LIN {X 0,Y 212.666,Z 436.056,A -85,B 0,C 180,E1 -21906.919,E2 -21906.919} C_VEL
LIN {X 0,Y 215.968,Z 426.694,A -85,B 0,C 180,E1 -21909.087,E2 -21909.087} C_VEL
LIN {X 0,Y 219.252,Z 415.76,A -85,B 0,C 180,E1 -21911.08,E2 -21911.08} C_VEL
LIN {X 0,Y 221.834,Z 405.227,A -85,B 0,C 180,E1 -21912.574,E2 -21912.574} C_VEL
LIN {X 0,Y 224.1,Z 393.658,A -85,B 0,C 180,E1 -21913.837,E2 -21913.837} C_VEL
LIN {X 0,Y 225.668,Z 381.684,A -85,B 0,C 180,E1 -21914.841,E2 -21914.841} C_VEL
LIN {X 0,Y 226.691,Z 369.485,A -85,B 0,C 180,E1 -21915.541,E2 -21915.541} C_VEL
LIN {X 0,Y 228.107,Z 336.25,A -85,B 0,C 180,E1 -21916.66,E2 -21916.66} C_VEL
LIN {X 0,Y 221.645,Z 324.171,A -85,B 0,C 180,E1 -21918.78,E2 -21918.78} C_VEL
LIN {X 0,Y 214.301,Z 312.104,A -85,B 0,C 180,E1 -21921.381,E2 -21921.381} C_VEL
LIN {X 0,Y 208.554,Z 303.596,A -85,B 0,C 180,E1 -21923.598,E2 -21923.598} C_VEL
LIN {X 0,Y 205.749,Z 299.629,A -85,B 0,C 180,E1 -21924.755,E2 -21924.755} C_VEL
LIN {X 0,Y 203.216,Z 296.188,A -85,B 0,C 180,E1 -21925.848,E2 -21925.848} C_VEL
LIN {X 0,Y 200.594,Z 292.5,A -85,B 0,C 180,E1 -21927.048,E2 -21927.048} C_VEL
LIN {X 0,Y 197.526,Z 288.904,A -85,B 0,C 180,E1 -21928.494,E2 -21928.494} C_VEL
LIN {X 0,Y 196.478,Z 286.965,A -85,B 0,C 180,E1 -21929.056,E2 -21929.056} C_VEL
LIN {X 0,Y 193.88,Z 284.765,A -85,B 0,C 180,E1 -21930.338,E2 -21930.338} C_VEL
LIN {X 0,Y 192.729,Z 282.176,A -85,B 0,C 180,E1 -21931.187,E2 -21931.187} C_VEL
LIN {X 0,Y 192.614,Z 281.525,A -85,B 0,C 180,E1 -21931.979,E2 -21931.979} C_VEL
LIN {X 0,Y 192.678,Z 281.429,A -85,B 0,C 180,E1 -21936.344,E2 -21936.344} C_VEL
LIN {X 0,Y 192.731,Z 281.449,A -85,B 0,C 180,E1 -21941.459,E2 -21941.459} C_VEL
LIN {X 0,Y 192.761,Z 281.455,A -85,B 0,C 180,E1 -21945.213,E2 -21945.213} C_VEL
LIN {X 0,Y 192.945,Z 281.435,A -85,B 0,C 180,E1 -21949.566,E2 -21949.566} C_VEL
LIN {X 0,Y 192.961,Z 281.448,A -85,B 0,C 180,E1 -21953.727,E2 -21953.727} C_VEL
LIN {X 0,Y 193.226,Z 281.405,A -85,B 0,C 180,E1 -21957.915,E2 -21957.915} C_VEL
LIN {X 0,Y 193.411,Z 281.384,A -85,B 0,C 180,E1 -21960,E2 -21960} C_VEL
LIN {X 0,Y 192.936,Z 281.449,A -85,B 0,C 180,E1 -21964.177,E2 -21964.177} C_VEL
LIN {X 0,Y 193.019,Z 281.422,A -85,B 0,C 180,E1 -21968.374,E2 -21968.374} C_VEL
LIN {X 0,Y 192.791,Z 281.45,A -85,B 0,C 180,E1 -21972.634,E2 -21972.634} C_VEL
LIN {X 0,Y 192.745,Z 281.468,A -85,B 0,C 180,E1 -21976.959,E2 -21976.959} C_VEL
LIN {X 0,Y 192.607,Z 281.485,A -85,B 0,C 180,E1 -21981.4,E2 -21981.4} C_VEL
LIN {X 0,Y 192.637,Z 281.491,A -85,B 0,C 180,E1 -21984.207,E2 -21984.207} C_VEL
LIN {X 0,Y 192.59,Z 281.62,A -85,B 0,C 180,E1 -21989.237,E2 -21989.237} C_VEL
LIN {X 0,Y 195.024,Z 288.184,A -85,B 0,C 180,E1 -21994.021,E2 -21994.021} C_VEL
LIN {X 0,Y 197.384,Z 295.043,A -85,B 0,C 180,E1 -21998.172,E2 -21998.172} C_VEL
LIN {X 0,Y 200.88,Z 300.852,A -85,B 0,C 180,E1 -21999.925,E2 -21999.925} C_VEL
LIN {X 0,Y 205.909,Z 309.501,A -85,B 0,C 180,E1 -22002.219,E2 -22002.219} C_VEL
LIN {X 0,Y 211.718,Z 320.154,A -85,B 0,C 180,E1 -22004.642,E2 -22004.642} C_VEL
LIN {X 0,Y 218.15,Z 333.803,A -85,B 0,C 180,E1 -22007.132,E2 -22007.132} C_VEL
LIN {X 0,Y 221.255,Z 341.29,A -85,B 0,C 180,E1 -22008.283,E2 -22008.283} C_VEL
LIN {X 0,Y 223.88,Z 365.922,A -85,B 0,C 180,E1 -22010.005,E2 -22010.005} C_VEL
LIN {X 0,Y 225.176,Z 381.652,A -85,B 0,C 180,E1 -22010.974,E2 -22010.974} C_VEL
LIN {X 0,Y 225.14,Z 385.521,A -85,B 0,C 180,E1 -22011.123,E2 -22011.123} C_VEL
LIN {X 0,Y 224.591,Z 389.408,A -85,B 0,C 180,E1 -22011.15,E2 -22011.15} C_VEL
LIN {X 0,Y 222.563,Z 397.072,A -85,B 0,C 180,E1 -22010.993,E2 -22010.993} C_VEL
LIN {X 0,Y 219.634,Z 406.689,A -85,B 0,C 180,E1 -22010.771,E2 -22010.771} C_VEL
LIN {X 0,Y 218.506,Z 412.571,A -85,B 0,C 180,E1 -22010.868,E2 -22010.868} C_VEL
LIN {X 0,Y 216.715,Z 425.149,A -85,B 0,C 180,E1 -22011.544,E2 -22011.544} C_VEL
LIN {X 0,Y 214.369,Z 437.19,A -85,B 0,C 180,E1 -22012.514,E2 -22012.514} C_VEL
LIN {X 0,Y 211.274,Z 449.041,A -85,B 0,C 180,E1 -22013.811,E2 -22013.811} C_VEL
LIN {X 0,Y 207.43,Z 460.468,A -85,B 0,C 180,E1 -22015.423,E2 -22015.423} C_VEL
LIN {X 0,Y 203.471,Z 470.808,A -85,B 0,C 180,E1 -22017.337,E2 -22017.337} C_VEL
LIN {X 0,Y 199.84,Z 479.297,A -85,B 0,C 180,E1 -22019.34,E2 -22019.34} C_VEL
LIN {X 0,Y 195.583,Z 488.554,A -85,B 0,C 180,E1 -22022.151,E2 -22022.151} C_VEL
LIN {X 0,Y 191.938,Z 496.066,A -85,B 0,C 180,E1 -22025.097,E2 -22025.097} C_VEL
LIN {X 0,Y 189.021,Z 502.163,A -85,B 0,C 180,E1 -22028.172,E2 -22028.172} C_VEL
LIN {X 0,Y 186.746,Z 507.041,A -85,B 0,C 180,E1 -22031.343,E2 -22031.343} C_VEL
LIN {X 0,Y 185.142,Z 510.839,A -85,B 0,C 180,E1 -22034.59,E2 -22034.59} C_VEL
LIN {X 0,Y 184.418,Z 512.843,A -85,B 0,C 180,E1 -22036.781,E2 -22036.781} C_VEL
LIN {X 0,Y 183.924,Z 515.566,A -85,B 0,C 180,E1 -22041.207,E2 -22041.207} C_VEL
LIN {X 0,Y 184.069,Z 516.35,A -85,B 0,C 180,E1 -22043.422,E2 -22043.422} C_VEL
LIN {X 0,Y 184.377,Z 516.743,A -85,B 0,C 180,E1 -22045.627,E2 -22045.627} C_VEL
LIN {X 0,Y 184.782,Z 516.697,A -85,B 0,C 180,E1 -22047.819,E2 -22047.819} C_VEL
LIN {X 0,Y 184.966,Z 516.195,A -85,B 0,C 180,E1 -22049.999,E2 -22049.999} C_VEL
LIN {X 0,Y 184.839,Z 515.234,A -85,B 0,C 180,E1 -22052.178,E2 -22052.178} C_VEL
LIN {X 0,Y 184.476,Z 513.812,A -85,B 0,C 180,E1 -22054.369,E2 -22054.369} C_VEL
LIN {X 0,Y 184.149,Z 511.34,A -85,B 0,C 180,E1 -22057.124,E2 -22057.124} C_VEL
LIN {X 0,Y 184.126,Z 506.671,A -85,B 0,C 180,E1 -22061.001,E2 -22061.001} C_VEL
LIN {X 0,Y 184.943,Z 500.384,A -85,B 0,C 180,E1 -22064.862,E2 -22064.862} C_VEL
LIN {X 0,Y 186.225,Z 493.516,A -85,B 0,C 180,E1 -22068.139,E2 -22068.139} C_VEL
LIN {X 0,Y 188.344,Z 485.062,A -85,B 0,C 180,E1 -22071.332,E2 -22071.332} C_VEL
LIN {X 0,Y 190.565,Z 476.381,A -85,B 0,C 180,E1 -22073.932,E2 -22073.932} C_VEL
LIN {X 0,Y 192.892,Z 466.861,A -85,B 0,C 180,E1 -22076.215,E2 -22076.215} C_VEL
LIN {X 0,Y 195.38,Z 456.548,A -85,B 0,C 180,E1 -22078.17,E2 -22078.17} C_VEL
LIN {X 0,Y 197.726,Z 445.275,A -85,B 0,C 180,E1 -22079.841,E2 -22079.841} C_VEL
LIN {X 0,Y 199.823,Z 432.646,A -85,B 0,C 180,E1 -22081.248,E2 -22081.248} C_VEL
LIN {X 0,Y 201.398,Z 419.7,A -85,B 0,C 180,E1 -22082.25,E2 -22082.25} C_VEL
LIN {X 0,Y 202.32,Z 405.805,A -85,B 0,C 180,E1 -22082.937,E2 -22082.937} C_VEL
LIN {X 0,Y 203.183,Z 381.621,A -85,B 0,C 180,E1 -22083.764,E2 -22083.764} C_VEL
LIN {X 0,Y 200.75,Z 344.71,A -85,B 0,C 180,E1 -22085.66,E2 -22085.66} C_VEL
LIN {X 0,Y 198.453,Z 320.123,A -85,B 0,C 180,E1 -22087.091,E2 -22087.091} C_VEL
LIN {X 0,Y 192.76,Z 305.892,A -85,B 0,C 180,E1 -22088.801,E2 -22088.801} C_VEL
LIN {X 0,Y 190.025,Z 299.446,A -85,B 0,C 180,E1 -22089.732,E2 -22089.732} C_VEL
LIN {X 0,Y 187.903,Z 291.059,A -85,B 0,C 180,E1 -22093.323,E2 -22093.323} C_VEL
LIN {X 0,Y 185.455,Z 282.487,A -85,B 0,C 180,E1 -22097.48,E2 -22097.48} C_VEL
LIN {X 0,Y 185.495,Z 282.366,A -85,B 0,C 180,E1 -22102.713,E2 -22102.713} C_VEL
LIN {X 0,Y 185.524,Z 282.35,A -85,B 0,C 180,E1 -22107.972,E2 -22107.972} C_VEL
LIN {X 0,Y 185.541,Z 282.371,A -85,B 0,C 180,E1 -22110.595,E2 -22110.595} C_VEL
LIN {X 0,Y 185.574,Z 282.351,A -85,B 0,C 180,E1 -22115.381,E2 -22115.381} C_VEL
LIN {X 0,Y 185.618,Z 282.342,A -85,B 0,C 180,E1 -22121.179,E2 -22121.179} C_VEL
LIN {X 0,Y 185.656,Z 282.353,A -85,B 0,C 180,E1 -22124.634,E2 -22124.634} C_VEL
LIN {X 0,Y 185.881,Z 282.307,A -85,B 0,C 180,E1 -22129.419,E2 -22129.419} C_VEL
LIN {X 0,Y 185.921,Z 282.323,A -85,B 0,C 180,E1 -22133.489,E2 -22133.489} C_VEL
LIN {X 0,Y 186.168,Z 282.272,A -85,B 0,C 180,E1 -22137.837,E2 -22137.837} C_VEL
LIN {X 0,Y 186.37,Z 282.242,A -85,B 0,C 180,E1 -22140,E2 -22140} C_VEL
LIN {X 0,Y 185.867,Z 282.333,A -85,B 0,C 180,E1 -22144.338,E2 -22144.338} C_VEL
LIN {X 0,Y 185.961,Z 282.291,A -85,B 0,C 180,E1 -22148.695,E2 -22148.695} C_VEL
LIN {X 0,Y 185.707,Z 282.35,A -85,B 0,C 180,E1 -22153.125,E2 -22153.125} C_VEL
LIN {X 0,Y 185.646,Z 282.33,A -85,B 0,C 180,E1 -22157.63,E2 -22157.63} C_VEL
LIN {X 0,Y 185.541,Z 282.373,A -85,B 0,C 180,E1 -22162.259,E2 -22162.259} C_VEL
LIN {X 0,Y 185.484,Z 282.36,A -85,B 0,C 180,E1 -22167.045,E2 -22167.045} C_VEL
LIN {X 0,Y 185.525,Z 282.363,A -85,B 0,C 180,E1 -22172.029,E2 -22172.029} C_VEL
LIN {X 0,Y 185.496,Z 282.38,A -85,B 0,C 180,E1 -22177.316,E2 -22177.316} C_VEL
LIN {X 0,Y 185.457,Z 282.336,A -85,B 0,C 180,E1 -22180.722,E2 -22180.722} C_VEL
LIN {X 0,Y 185.452,Z 282.349,A -85,B 0,C 180,E1 -22186.058,E2 -22186.058} C_VEL
LIN {X 0,Y 185.454,Z 282.367,A -85,B 0,C 180,E1 -22189.894,E2 -22189.894} C_VEL
LIN {X 0,Y 185.499,Z 282.332,A -85,B 0,C 180,E1 -22192.716,E2 -22192.716} C_VEL
LIN {X 0,Y 185.528,Z 282.48,A -85,B 0,C 180,E1 -22197.974,E2 -22197.974} C_VEL
LIN {X 0,Y 185.696,Z 283.33,A -85,B 0,C 180,E1 -22198.372,E2 -22198.372} C_VEL
LIN {X 0,Y 187.12,Z 286.075,A -85,B 0,C 180,E1 -22198.87,E2 -22198.87} C_VEL
LIN {X 0,Y 190.505,Z 291.53,A -85,B 0,C 180,E1 -22199.867,E2 -22199.867} C_VEL
LIN {X 0,Y 196.709,Z 302.532,A -85,B 0,C 180,E1 -22201.62,E2 -22201.62} C_VEL
LIN {X 0,Y 203.781,Z 317.099,A -85,B 0,C 180,E1 -22203.532,E2 -22203.532} C_VEL
LIN {X 0,Y 205.564,Z 321.268,A -85,B 0,C 180,E1 -22204.008,E2 -22204.008} C_VEL
LIN {X 0,Y 204.008,Z 369.15,A -85,B 0,C 180,E1 -22205.719,E2 -22205.719} C_VEL
LIN {X 0,Y 203.326,Z 380.674,A -85,B 0,C 180,E1 -22206.445,E2 -22206.445} C_VEL
LIN {X 0,Y 202.053,Z 393.603,A -85,B 0,C 180,E1 -22207.641,E2 -22207.641} C_VEL
LIN {X 0,Y 200.279,Z 405.935,A -85,B 0,C 180,E1 -22209.19,E2 -22209.19} C_VEL
LIN {X 0,Y 198.141,Z 417.489,A -85,B 0,C 180,E1 -22211.117,E2 -22211.117} C_VEL
LIN {X 0,Y 195.987,Z 427.846,A -85,B 0,C 180,E1 -22213.33,E2 -22213.33} C_VEL
LIN {X 0,Y 193.789,Z 437.202,A -85,B 0,C 180,E1 -22215.831,E2 -22215.831} C_VEL
LIN {X 0,Y 191.383,Z 446.228,A -85,B 0,C 180,E1 -22218.885,E2 -22218.885} C_VEL
LIN {X 0,Y 189.347,Z 453.509,A -85,B 0,C 180,E1 -22222,E2 -22222} C_VEL
LIN {X 0,Y 187.582,Z 460.199,A -85,B 0,C 180,E1 -22225.704,E2 -22225.704} C_VEL
LIN {X 0,Y 186.487,Z 464.627,A -85,B 0,C 180,E1 -22228.921,E2 -22228.921} C_VEL
LIN {X 0,Y 185.647,Z 468.025,A -85,B 0,C 180,E1 -22232.17,E2 -22232.17} C_VEL
LIN {X 0,Y 185.454,Z 470.993,A -85,B 0,C 180,E1 -22236.529,E2 -22236.529} C_VEL
LIN {X 0,Y 185.694,Z 472.291,A -85,B 0,C 180,E1 -22240.25,E2 -22240.25} C_VEL
LIN {X 0,Y 186.169,Z 472.505,A -85,B 0,C 180,E1 -22243.092,E2 -22243.092} C_VEL
LIN {X 0,Y 187.574,Z 471.565,A -85,B 0,C 180,E1 -22247.443,E2 -22247.443} C_VEL
LIN {X 0,Y 188.562,Z 470.463,A -85,B 0,C 180,E1 -22249.6,E2 -22249.6} C_VEL
LIN {X 0,Y 190.407,Z 468.162,A -85,B 0,C 180,E1 -22252.665,E2 -22252.665} C_VEL
LIN {X 0,Y 192.795,Z 464.602,A -85,B 0,C 180,E1 -22255.941,E2 -22255.941} C_VEL
LIN {X 0,Y 195.549,Z 460.037,A -85,B 0,C 180,E1 -22259.025,E2 -22259.025} C_VEL
LIN {X 0,Y 199.375,Z 453.086,A -85,B 0,C 180,E1 -22262.518,E2 -22262.518} C_VEL
LIN {X 0,Y 203.086,Z 445.472,A -85,B 0,C 180,E1 -22265.426,E2 -22265.426} C_VEL
LIN {X 0,Y 206.92,Z 436.495,A -85,B 0,C 180,E1 -22268.074,E2 -22268.074} C_VEL
LIN {X 0,Y 210.426,Z 426.876,A -85,B 0,C 180,E1 -22270.324,E2 -22270.324} C_VEL
LIN {X 0,Y 213.492,Z 417.125,A -85,B 0,C 180,E1 -22272.123,E2 -22272.123} C_VEL
LIN {X 0,Y 216.14,Z 406.913,A -85,B 0,C 180,E1 -22273.623,E2 -22273.623} C_VEL
LIN {X 0,Y 218.749,Z 394.311,A -85,B 0,C 180,E1 -22275.022,E2 -22275.022} C_VEL
LIN {X 0,Y 220.418,Z 381.923,A -85,B 0,C 180,E1 -22276.072,E2 -22276.072} C_VEL
LIN {X 0,Y 221.447,Z 369.834,A -85,B 0,C 180,E1 -22276.763,E2 -22276.763} C_VEL
LIN {X 0,Y 222.794,Z 338.838,A -85,B 0,C 180,E1 -22277.833,E2 -22277.833} C_VEL
LIN {X 0,Y 216.755,Z 327.518,A -85,B 0,C 180,E1 -22279.939,E2 -22279.939} C_VEL
LIN {X 0,Y 210.199,Z 316.66,A -85,B 0,C 180,E1 -22282.396,E2 -22282.396} C_VEL
LIN {X 0,Y 204.778,Z 308.452,A -85,B 0,C 180,E1 -22284.608,E2 -22284.608} C_VEL
LIN {X 0,Y 200.168,Z 301.967,A -85,B 0,C 180,E1 -22286.653,E2 -22286.653} C_VEL
LIN {X 0,Y 196.875,Z 297.515,A -85,B 0,C 180,E1 -22288.227,E2 -22288.227} C_VEL
LIN {X 0,Y 194.242,Z 294.054,A -85,B 0,C 180,E1 -22289.565,E2 -22289.565} C_VEL
LIN {X 0,Y 193.394,Z 292.857,A -85,B 0,C 180,E1 -22290.02,E2 -22290.02} C_VEL
LIN {X 0,Y 191.007,Z 290.431,A -85,B 0,C 180,E1 -22291.287,E2 -22291.287} C_VEL
LIN {X 0,Y 189.674,Z 287.958,A -85,B 0,C 180,E1 -22292.108,E2 -22292.108} C_VEL
LIN {X 0,Y 187.145,Z 286.062,A -85,B 0,C 180,E1 -22293.545,E2 -22293.545} C_VEL
LIN {X 0,Y 185.716,Z 283.299,A -85,B 0,C 180,E1 -22294.62,E2 -22294.62} C_VEL
LIN {X 0,Y 185.594,Z 282.426,A -85,B 0,C 180,E1 -22295.486,E2 -22295.486} C_VEL
LIN {X 0,Y 185.673,Z 282.318,A -85,B 0,C 180,E1 -22301.135,E2 -22301.135} C_VEL
LIN {X 0,Y 185.693,Z 282.337,A -85,B 0,C 180,E1 -22304.636,E2 -22304.636} C_VEL
LIN {X 0,Y 185.888,Z 282.315,A -85,B 0,C 180,E1 -22309.419,E2 -22309.419} C_VEL
LIN {X 0,Y 185.926,Z 282.326,A -85,B 0,C 180,E1 -22313.488,E2 -22313.488} C_VEL
LIN {X 0,Y 186.172,Z 282.282,A -85,B 0,C 180,E1 -22317.836,E2 -22317.836} C_VEL
LIN {X 0,Y 186.377,Z 282.26,A -85,B 0,C 180,E1 -22320,E2 -22320} C_VEL
LIN {X 0,Y 185.884,Z 282.329,A -85,B 0,C 180,E1 -22324.336,E2 -22324.336} C_VEL
LIN {X 0,Y 185.969,Z 282.302,A -85,B 0,C 180,E1 -22328.694,E2 -22328.694} C_VEL
LIN {X 0,Y 185.718,Z 282.33,A -85,B 0,C 180,E1 -22333.123,E2 -22333.123} C_VEL
LIN {X 0,Y 185.682,Z 282.344,A -85,B 0,C 180,E1 -22337.625,E2 -22337.625} C_VEL
LIN {X 0,Y 185.569,Z 282.36,A -85,B 0,C 180,E1 -22342.254,E2 -22342.254} C_VEL
LIN {X 0,Y 185.545,Z 282.567,A -85,B 0,C 180,E1 -22346.426,E2 -22346.426} C_VEL
LIN {X 0,Y 187.951,Z 288.856,A -85,B 0,C 180,E1 -22351.567,E2 -22351.567} C_VEL
LIN {X 0,Y 189.577,Z 293.321,A -85,B 0,C 180,E1 -22354.556,E2 -22354.556} C_VEL
LIN {X 0,Y 193.718,Z 299.814,A -85,B 0,C 180,E1 -22356.944,E2 -22356.944} C_VEL
LIN {X 0,Y 199.001,Z 308.663,A -85,B 0,C 180,E1 -22359.669,E2 -22359.669} C_VEL
LIN {X 0,Y 202.611,Z 315.139,A -85,B 0,C 180,E1 -22361.383,E2 -22361.383} C_VEL
LIN {X 0,Y 207.767,Z 324.854,A -85,B 0,C 180,E1 -22363.652,E2 -22363.652} C_VEL
LIN {X 0,Y 213.978,Z 338.398,A -85,B 0,C 180,E1 -22366.198,E2 -22366.198} C_VEL
LIN {X 0,Y 216.453,Z 344.843,A -85,B 0,C 180,E1 -22367.187,E2 -22367.187} C_VEL
LIN {X 0,Y 218.786,Z 368.364,A -85,B 0,C 180,E1 -22368.869,E2 -22368.869} C_VEL
LIN {X 0,Y 220.155,Z 387.448,A -85,B 0,C 180,E1 -22370.049,E2 -22370.049} C_VEL
LIN {X 0,Y 218.626,Z 411.388,A -85,B 0,C 180,E1 -22370.816,E2 -22370.816} C_VEL
LIN {X 0,Y 218.506,Z 412.571,A -85,B 0,C 180,E1 -22370.868,E2 -22370.868} C_VEL
LIN {X 0,Y 217.532,Z 416.438,A -85,B 0,C 180,E1 -22370.922,E2 -22370.922} C_VEL
LIN {X 0,Y 214.526,Z 422.459,A -85,B 0,C 180,E1 -22370.763,E2 -22370.763} C_VEL
LIN {X 0,Y 211.291,Z 428.377,A -85,B 0,C 180,E1 -22370.669,E2 -22370.669} C_VEL
LIN {X 0,Y 209.961,Z 432.081,A -85,B 0,C 180,E1 -22370.846,E2 -22370.846} C_VEL
LIN {X 0,Y 207.055,Z 443.97,A -85,B 0,C 180,E1 -22372.033,E2 -22372.033} C_VEL
LIN {X 0,Y 203.107,Z 456.364,A -85,B 0,C 180,E1 -22373.661,E2 -22373.661} C_VEL
LIN {X 0,Y 198.855,Z 467.265,A -85,B 0,C 180,E1 -22375.564,E2 -22375.564} C_VEL
LIN {X 0,Y 194.521,Z 477.091,A -85,B 0,C 180,E1 -22377.797,E2 -22377.797} C_VEL
LIN {X 0,Y 190.756,Z 485.197,A -85,B 0,C 180,E1 -22380.173,E2 -22380.173} C_VEL
LIN {X 0,Y 186.695,Z 493.199,A -85,B 0,C 180,E1 -22383.145,E2 -22383.145} C_VEL
LIN {X 0,Y 183.406,Z 499.661,A -85,B 0,C 180,E1 -22386.274,E2 -22386.274} C_VEL
LIN {X 0,Y 180.655,Z 504.858,A -85,B 0,C 180,E1 -22389.504,E2 -22389.504} C_VEL
LIN {X 0,Y 178.772,Z 508.973,A -85,B 0,C 180,E1 -22392.851,E2 -22392.851} C_VEL
LIN {X 0,Y 177.443,Z 512.076,A -85,B 0,C 180,E1 -22396.252,E2 -22396.252} C_VEL
LIN {X 0,Y 176.844,Z 514.752,A -85,B 0,C 180,E1 -22400.852,E2 -22400.852} C_VEL
LIN {X 0,Y 177,Z 515.522,A -85,B 0,C 180,E1 -22403.158,E2 -22403.158} C_VEL
LIN {X 0,Y 177.275,Z 515.887,A -85,B 0,C 180,E1 -22405.451,E2 -22405.451} C_VEL
LIN {X 0,Y 177.719,Z 515.816,A -85,B 0,C 180,E1 -22407.733,E2 -22407.733} C_VEL
LIN {X 0,Y 177.919,Z 515.297,A -85,B 0,C 180,E1 -22409.999,E2 -22409.999} C_VEL
LIN {X 0,Y 177.744,Z 514.31,A -85,B 0,C 180,E1 -22412.265,E2 -22412.265} C_VEL
LIN {X 0,Y 177.367,Z 512.856,A -85,B 0,C 180,E1 -22414.544,E2 -22414.544} C_VEL
LIN {X 0,Y 177.023,Z 509.787,A -85,B 0,C 180,E1 -22417.985,E2 -22417.985} C_VEL
LIN {X 0,Y 177.103,Z 505.63,A -85,B 0,C 180,E1 -22421.443,E2 -22421.443} C_VEL
LIN {X 0,Y 178.011,Z 499.269,A -85,B 0,C 180,E1 -22425.454,E2 -22425.454} C_VEL
LIN {X 0,Y 179.436,Z 492.349,A -85,B 0,C 180,E1 -22428.851,E2 -22428.851} C_VEL
LIN {X 0,Y 181.695,Z 483.732,A -85,B 0,C 180,E1 -22432.185,E2 -22432.185} C_VEL
LIN {X 0,Y 184.039,Z 475.033,A -85,B 0,C 180,E1 -22434.837,E2 -22434.837} C_VEL
LIN {X 0,Y 186.439,Z 465.402,A -85,B 0,C 180,E1 -22437.196,E2 -22437.196} C_VEL
LIN {X 0,Y 188.767,Z 456.418,A -85,B 0,C 180,E1 -22438.945,E2 -22438.945} C_VEL
LIN {X 0,Y 191.208,Z 445.319,A -85,B 0,C 180,E1 -22440.661,E2 -22440.661} C_VEL
LIN {X 0,Y 193.38,Z 433.007,A -85,B 0,C 180,E1 -22442.106,E2 -22442.106} C_VEL
LIN {X 0,Y 195.043,Z 420.403,A -85,B 0,C 180,E1 -22443.151,E2 -22443.151} C_VEL
LIN {X 0,Y 196.029,Z 407.345,A -85,B 0,C 180,E1 -22443.859,E2 -22443.859} C_VEL
LIN {X 0,Y 197.053,Z 382.986,A -85,B 0,C 180,E1 -22444.714,E2 -22444.714} C_VEL
LIN {X 0,Y 194.738,Z 345.918,A -85,B 0,C 180,E1 -22446.685,E2 -22446.685} C_VEL
LIN {X 0,Y 192.633,Z 322.522,A -85,B 0,C 180,E1 -22448.097,E2 -22448.097} C_VEL
LIN {X 0,Y 186.404,Z 306.851,A -85,B 0,C 180,E1 -22450.098,E2 -22450.098} C_VEL
LIN {X 0,Y 182.658,Z 298.536,A -85,B 0,C 180,E1 -22451.405,E2 -22451.405} C_VEL
LIN {X 0,Y 180.871,Z 291.89,A -85,B 0,C 180,E1 -22454.378,E2 -22454.378} C_VEL
LIN {X 0,Y 178.422,Z 283.367,A -85,B 0,C 180,E1 -22458.748,E2 -22458.748} C_VEL
LIN {X 0,Y 178.413,Z 283.259,A -85,B 0,C 180,E1 -22463.781,E2 -22463.781} C_VEL
LIN {X 0,Y 178.478,Z 283.23,A -85,B 0,C 180,E1 -22466.545,E2 -22466.545} C_VEL
LIN {X 0,Y 178.437,Z 283.258,A -85,B 0,C 180,E1 -22471.795,E2 -22471.795} C_VEL
LIN {X 0,Y 178.509,Z 283.228,A -85,B 0,C 180,E1 -22474.889,E2 -22474.889} C_VEL
LIN {X 0,Y 178.6,Z 283.213,A -85,B 0,C 180,E1 -22481.651,E2 -22481.651} C_VEL
LIN {X 0,Y 178.634,Z 283.234,A -85,B 0,C 180,E1 -22486.346,E2 -22486.346} C_VEL
LIN {X 0,Y 178.896,Z 283.174,A -85,B 0,C 180,E1 -22490.959,E2 -22490.959} C_VEL
LIN {X 0,Y 179.116,Z 283.15,A -85,B 0,C 180,E1 -22497.752,E2 -22497.752} C_VEL
LIN {X 0,Y 179.335,Z 283.117,A -85,B 0,C 180,E1 -22500,E2 -22500} C_VEL
LIN {X 0,Y 178.816,Z 283.21,A -85,B 0,C 180,E1 -22504.509,E2 -22504.509} C_VEL
LIN {X 0,Y 178.894,Z 283.17,A -85,B 0,C 180,E1 -22509.042,E2 -22509.042} C_VEL
LIN {X 0,Y 178.634,Z 283.232,A -85,B 0,C 180,E1 -22513.655,E2 -22513.655} C_VEL
LIN {X 0,Y 178.549,Z 283.222,A -85,B 0,C 180,E1 -22519.154,E2 -22519.154} C_VEL
LIN {X 0,Y 178.458,Z 283.232,A -85,B 0,C 180,E1 -22525.077,E2 -22525.077} C_VEL
LIN {X 0,Y 178.445,Z 283.255,A -85,B 0,C 180,E1 -22530.798,E2 -22530.798} C_VEL
LIN {X 0,Y 178.478,Z 283.233,A -85,B 0,C 180,E1 -22534.219,E2 -22534.219} C_VEL
LIN {X 0,Y 178.382,Z 283.247,A -85,B 0,C 180,E1 -22539.079,E2 -22539.079} C_VEL
LIN {X 0,Y 178.389,Z 283.198,A -85,B 0,C 180,E1 -22542.049,E2 -22542.049} C_VEL
LIN {X 0,Y 178.388,Z 283.21,A -85,B 0,C 180,E1 -22545.167,E2 -22545.167} C_VEL
LIN {X 0,Y 178.395,Z 283.265,A -85,B 0,C 180,E1 -22548.463,E2 -22548.463} C_VEL
LIN {X 0,Y 178.417,Z 283.216,A -85,B 0,C 180,E1 -22553.784,E2 -22553.784} C_VEL
LIN {X 0,Y 178.519,Z 283.518,A -85,B 0,C 180,E1 -22556.417,E2 -22556.417} C_VEL
LIN {X 0,Y 178.889,Z 284.831,A -85,B 0,C 180,E1 -22556.821,E2 -22556.821} C_VEL
LIN {X 0,Y 180.617,Z 287.486,A -85,B 0,C 180,E1 -22557.401,E2 -22557.401} C_VEL
LIN {X 0,Y 188.928,Z 301.506,A -85,B 0,C 180,E1 -22559.984,E2 -22559.984} C_VEL
LIN {X 0,Y 196.997,Z 317.521,A -85,B 0,C 180,E1 -22562.318,E2 -22562.318} C_VEL
LIN {X 0,Y 199.474,Z 323.359,A -85,B 0,C 180,E1 -22563.024,E2 -22563.024} C_VEL
LIN {X 0,Y 197.795,Z 370.595,A -85,B 0,C 180,E1 -22564.763,E2 -22564.763} C_VEL
LIN {X 0,Y 197.092,Z 381.91,A -85,B 0,C 180,E1 -22565.512,E2 -22565.512} C_VEL
LIN {X 0,Y 195.748,Z 394.738,A -85,B 0,C 180,E1 -22566.74,E2 -22566.74} C_VEL
LIN {X 0,Y 194.04,Z 406.146,A -85,B 0,C 180,E1 -22568.209,E2 -22568.209} C_VEL
LIN {X 0,Y 191.798,Z 417.86,A -85,B 0,C 180,E1 -22570.189,E2 -22570.189} C_VEL
LIN {X 0,Y 189.536,Z 428.297,A -85,B 0,C 180,E1 -22572.467,E2 -22572.467} C_VEL
LIN {X 0,Y 186.986,Z 438.57,A -85,B 0,C 180,E1 -22575.304,E2 -22575.304} C_VEL
LIN {X 0,Y 184.474,Z 447.497,A -85,B 0,C 180,E1 -22578.464,E2 -22578.464} C_VEL
LIN {X 0,Y 182.388,Z 454.701,A -85,B 0,C 180,E1 -22581.693,E2 -22581.693} C_VEL
LIN {X 0,Y 181.06,Z 459.572,A -85,B 0,C 180,E1 -22584.432,E2 -22584.432} C_VEL
LIN {X 0,Y 179.761,Z 464.328,A -85,B 0,C 180,E1 -22587.76,E2 -22587.76} C_VEL
LIN {X 0,Y 178.814,Z 468.004,A -85,B 0,C 180,E1 -22591.127,E2 -22591.127} C_VEL
LIN {X 0,Y 178.423,Z 470.667,A -85,B 0,C 180,E1 -22594.519,E2 -22594.519} C_VEL
LIN {X 0,Y 178.41,Z 471.933,A -85,B 0,C 180,E1 -22596.788,E2 -22596.788} C_VEL
LIN {X 0,Y 178.674,Z 473.139,A -85,B 0,C 180,E1 -22600.464,E2 -22600.464} C_VEL
LIN {X 0,Y 179.237,Z 473.348,A -85,B 0,C 180,E1 -22603.608,E2 -22603.608} C_VEL
LIN {X 0,Y 179.911,Z 473.045,A -85,B 0,C 180,E1 -22605.87,E2 -22605.87} C_VEL
LIN {X 0,Y 180.778,Z 472.346,A -85,B 0,C 180,E1 -22608.121,E2 -22608.121} C_VEL
LIN {X 0,Y 181.855,Z 471.206,A -85,B 0,C 180,E1 -22610.354,E2 -22610.354} C_VEL
LIN {X 0,Y 183.682,Z 469.046,A -85,B 0,C 180,E1 -22613.321,E2 -22613.321} C_VEL
LIN {X 0,Y 186.393,Z 465.236,A -85,B 0,C 180,E1 -22616.902,E2 -22616.902} C_VEL
LIN {X 0,Y 189.323,Z 460.61,A -85,B 0,C 180,E1 -22620.076,E2 -22620.076} C_VEL
LIN {X 0,Y 192.75,Z 454.697,A -85,B 0,C 180,E1 -22623.157,E2 -22623.157} C_VEL
LIN {X 0,Y 196.6,Z 447.279,A -85,B 0,C 180,E1 -22626.146,E2 -22626.146} C_VEL
LIN {X 0,Y 200.162,Z 439.645,A -85,B 0,C 180,E1 -22628.552,E2 -22628.552} C_VEL
LIN {X 0,Y 203.852,Z 430.268,A -85,B 0,C 180,E1 -22630.923,E2 -22630.923} C_VEL
LIN {X 0,Y 207.415,Z 419.763,A -85,B 0,C 180,E1 -22632.993,E2 -22632.993} C_VEL
LIN {X 0,Y 210.587,Z 408.315,A -85,B 0,C 180,E1 -22634.76,E2 -22634.76} C_VEL
LIN {X 0,Y 213.217,Z 396.321,A -85,B 0,C 180,E1 -22636.142,E2 -22636.142} C_VEL
LIN {X 0,Y 215.028,Z 384.131,A -85,B 0,C 180,E1 -22637.215,E2 -22637.215} C_VEL
LIN {X 0,Y 216.106,Z 373.156,A -85,B 0,C 180,E1 -22637.893,E2 -22637.893} C_VEL
LIN {X 0,Y 217.045,Z 354.634,A -85,B 0,C 180,E1 -22638.597,E2 -22638.597} C_VEL
LIN {X 0,Y 217.556,Z 341.405,A -85,B 0,C 180,E1 -22639.072,E2 -22639.072} C_VEL
LIN {X 0,Y 210.814,Z 328.836,A -85,B 0,C 180,E1 -22641.593,E2 -22641.593} C_VEL
LIN {X 0,Y 202.87,Z 315.926,A -85,B 0,C 180,E1 -22644.862,E2 -22644.862} C_VEL
LIN {X 0,Y 196.87,Z 307.354,A -85,B 0,C 180,E1 -22647.623,E2 -22647.623} C_VEL
LIN {X 0,Y 193.77,Z 303.143,A -85,B 0,C 180,E1 -22649.181,E2 -22649.181} C_VEL
LIN {X 0,Y 190.593,Z 298.893,A -85,B 0,C 180,E1 -22650.898,E2 -22650.898} C_VEL
LIN {X 0,Y 188.022,Z 295.765,A -85,B 0,C 180,E1 -22652.371,E2 -22652.371} C_VEL
LIN {X 0,Y 186.959,Z 294.17,A -85,B 0,C 180,E1 -22653.034,E2 -22653.034} C_VEL
LIN {X 0,Y 184.405,Z 291.722,A -85,B 0,C 180,E1 -22654.611,E2 -22654.611} C_VEL
LIN {X 0,Y 182.865,Z 288.946,A -85,B 0,C 180,E1 -22655.731,E2 -22655.731} C_VEL
LIN {X 0,Y 180.118,Z 286.805,A -85,B 0,C 180,E1 -22657.639,E2 -22657.639} C_VEL
LIN {X 0,Y 178.77,Z 284.422,A -85,B 0,C 180,E1 -22658.826,E2 -22658.826} C_VEL
LIN {X 0,Y 178.582,Z 283.45,A -85,B 0,C 180,E1 -22659.599,E2 -22659.599} C_VEL
LIN {X 0,Y 178.648,Z 283.202,A -85,B 0,C 180,E1 -22661.656,E2 -22661.656} C_VEL
LIN {X 0,Y 178.656,Z 283.214,A -85,B 0,C 180,E1 -22666.347,E2 -22666.347} C_VEL
LIN {X 0,Y 178.903,Z 283.179,A -85,B 0,C 180,E1 -22670.959,E2 -22670.959} C_VEL
LIN {X 0,Y 179.119,Z 283.159,A -85,B 0,C 180,E1 -22677.751,E2 -22677.751} C_VEL
LIN {X 0,Y 179.342,Z 283.135,A -85,B 0,C 180,E1 -22680,E2 -22680} C_VEL
LIN {X 0,Y 178.833,Z 283.209,A -85,B 0,C 180,E1 -22684.508,E2 -22684.508} C_VEL
LIN {X 0,Y 178.901,Z 283.185,A -85,B 0,C 180,E1 -22689.04,E2 -22689.04} C_VEL
LIN {X 0,Y 178.647,Z 283.211,A -85,B 0,C 180,E1 -22693.653,E2 -22693.653} C_VEL
LIN {X 0,Y 178.608,Z 283.23,A -85,B 0,C 180,E1 -22699.202,E2 -22699.202} C_VEL
LIN {X 0,Y 178.543,Z 283.423,A -85,B 0,C 180,E1 -22703.027,E2 -22703.027} C_VEL
LIN {X 0,Y 180.409,Z 288.564,A -85,B 0,C 180,E1 -22707.87,E2 -22707.87} C_VEL
LIN {X 0,Y 181.524,Z 291.333,A -85,B 0,C 180,E1 -22709.979,E2 -22709.979} C_VEL
LIN {X 0,Y 187.109,Z 299.664,A -85,B 0,C 180,E1 -22713.805,E2 -22713.805} C_VEL
LIN {X 0,Y 191.667,Z 307.029,A -85,B 0,C 180,E1 -22716.511,E2 -22716.511} C_VEL
LIN {X 0,Y 196.182,Z 314.871,A -85,B 0,C 180,E1 -22718.935,E2 -22718.935} C_VEL
LIN {X 0,Y 199.235,Z 320.508,A -85,B 0,C 180,E1 -22720.458,E2 -22720.458} C_VEL
LIN {X 0,Y 204.276,Z 330.42,A -85,B 0,C 180,E1 -22722.803,E2 -22722.803} C_VEL
LIN {X 0,Y 209.643,Z 342.407,A -85,B 0,C 180,E1 -22725.13,E2 -22725.13} C_VEL
LIN {X 0,Y 211.607,Z 347.396,A -85,B 0,C 180,E1 -22725.955,E2 -22725.955} C_VEL
LIN {X 0,Y 213.626,Z 368.549,A -85,B 0,C 180,E1 -22727.531,E2 -22727.531} C_VEL
LIN {X 0,Y 214.957,Z 387.567,A -85,B 0,C 180,E1 -22728.762,E2 -22728.762} C_VEL
LIN {X 0,Y 213.467,Z 410.427,A -85,B 0,C 180,E1 -22729.514,E2 -22729.514} C_VEL
LIN {X 0,Y 211.523,Z 424.033,A -85,B 0,C 180,E1 -22730.235,E2 -22730.235} C_VEL
LIN {X 0,Y 209.961,Z 432.081,A -85,B 0,C 180,E1 -22730.846,E2 -22730.846} C_VEL
LIN {X 0,Y 208.104,Z 437.7,A -85,B 0,C 180,E1 -22731.229,E2 -22731.229} C_VEL
LIN {X 0,Y 203.46,Z 446.41,A -85,B 0,C 180,E1 -22731.68,E2 -22731.68} C_VEL
LIN {X 0,Y 198.515,Z 454.585,A -85,B 0,C 180,E1 -22732.307,E2 -22732.307} C_VEL
LIN {X 0,Y 196.189,Z 459.393,A -85,B 0,C 180,E1 -22732.964,E2 -22732.964} C_VEL
LIN {X 0,Y 192.104,Z 469.094,A -85,B 0,C 180,E1 -22734.816,E2 -22734.816} C_VEL
LIN {X 0,Y 187.723,Z 478.412,A -85,B 0,C 180,E1 -22737.122,E2 -22737.122} C_VEL
LIN {X 0,Y 183.128,Z 487.52,A -85,B 0,C 180,E1 -22740.072,E2 -22740.072} C_VEL
LIN {X 0,Y 179.126,Z 494.911,A -85,B 0,C 180,E1 -22743.179,E2 -22743.179} C_VEL
LIN {X 0,Y 175.87,Z 500.897,A -85,B 0,C 180,E1 -22746.446,E2 -22746.446} C_VEL
LIN {X 0,Y 173.241,Z 505.67,A -85,B 0,C 180,E1 -22749.828,E2 -22749.828} C_VEL
LIN {X 0,Y 171.418,Z 509.384,A -85,B 0,C 180,E1 -22753.321,E2 -22753.321} C_VEL
LIN {X 0,Y 170.5,Z 511.305,A -85,B 0,C 180,E1 -22755.68,E2 -22755.68} C_VEL
LIN {X 0,Y 169.79,Z 513.94,A -85,B 0,C 180,E1 -22760.469,E2 -22760.469} C_VEL
LIN {X 0,Y 169.934,Z 514.729,A -85,B 0,C 180,E1 -22763.012,E2 -22763.012} C_VEL
LIN {X 0,Y 170.653,Z 514.935,A -85,B 0,C 180,E1 -22767.639,E2 -22767.639} C_VEL
LIN {X 0,Y 170.872,Z 514.4,A -85,B 0,C 180,E1 -22769.999,E2 -22769.999} C_VEL
LIN {X 0,Y 170.65,Z 513.386,A -85,B 0,C 180,E1 -22772.359,E2 -22772.359} C_VEL
LIN {X 0,Y 170.259,Z 511.892,A -85,B 0,C 180,E1 -22774.734,E2 -22774.734} C_VEL
LIN {X 0,Y 169.946,Z 508.784,A -85,B 0,C 180,E1 -22778.32,E2 -22778.32} C_VEL
LIN {X 0,Y 170.108,Z 504.582,A -85,B 0,C 180,E1 -22781.92,E2 -22781.92} C_VEL
LIN {X 0,Y 171.118,Z 498.155,A -85,B 0,C 180,E1 -22786.094,E2 -22786.094} C_VEL
LIN {X 0,Y 172.676,Z 491.178,A -85,B 0,C 180,E1 -22789.618,E2 -22789.618} C_VEL
LIN {X 0,Y 174.997,Z 482.709,A -85,B 0,C 180,E1 -22792.988,E2 -22792.988} C_VEL
LIN {X 0,Y 177.791,Z 472.674,A -85,B 0,C 180,E1 -22796.087,E2 -22796.087} C_VEL
LIN {X 0,Y 180.504,Z 462.773,A -85,B 0,C 180,E1 -22798.485,E2 -22798.485} C_VEL
LIN {X 0,Y 183.288,Z 451.932,A -85,B 0,C 180,E1 -22800.533,E2 -22800.533} C_VEL
LIN {X 0,Y 185.894,Z 439.746,A -85,B 0,C 180,E1 -22802.275,E2 -22802.275} C_VEL
LIN {X 0,Y 188.017,Z 427.006,A -85,B 0,C 180,E1 -22803.618,E2 -22803.618} C_VEL
LIN {X 0,Y 189.436,Z 414.04,A -85,B 0,C 180,E1 -22804.565,E2 -22804.565} C_VEL
LIN {X 0,Y 190.365,Z 398.289,A -85,B 0,C 180,E1 -22805.234,E2 -22805.234} C_VEL
LIN {X 0,Y 190.911,Z 382.796,A -85,B 0,C 180,E1 -22805.804,E2 -22805.804} C_VEL
LIN {X 0,Y 188.68,Z 346.238,A -85,B 0,C 180,E1 -22807.835,E2 -22807.835} C_VEL
LIN {X 0,Y 186.865,Z 324.85,A -85,B 0,C 180,E1 -22809.172,E2 -22809.172} C_VEL
LIN {X 0,Y 181.1,Z 310.273,A -85,B 0,C 180,E1 -22811.14,E2 -22811.14} C_VEL
LIN {X 0,Y 176.651,Z 300.828,A -85,B 0,C 180,E1 -22812.694,E2 -22812.694} C_VEL
LIN {X 0,Y 174.96,Z 296.948,A -85,B 0,C 180,E1 -22813.485,E2 -22813.485} C_VEL
LIN {X 0,Y 172.399,Z 287.851,A -85,B 0,C 180,E1 -22818.087,E2 -22818.087} C_VEL
LIN {X 0,Y 171.364,Z 284.226,A -85,B 0,C 180,E1 -22820.206,E2 -22820.206} C_VEL
LIN {X 0,Y 171.392,Z 284.129,A -85,B 0,C 180,E1 -22825.092,E2 -22825.092} C_VEL
LIN {X 0,Y 171.402,Z 284.132,A -85,B 0,C 180,E1 -22830.526,E2 -22830.526} C_VEL
LIN {X 0,Y 171.43,Z 284.113,A -85,B 0,C 180,E1 -22835.798,E2 -22835.798} C_VEL
LIN {X 0,Y 171.5,Z 284.1,A -85,B 0,C 180,E1 -22840.863,E2 -22840.863} C_VEL
LIN {X 0,Y 171.548,Z 284.116,A -85,B 0,C 180,E1 -22845.771,E2 -22845.771} C_VEL
LIN {X 0,Y 171.835,Z 284.051,A -85,B 0,C 180,E1 -22850.585,E2 -22850.585} C_VEL
LIN {X 0,Y 171.775,Z 284.087,A -85,B 0,C 180,E1 -22855.307,E2 -22855.307} C_VEL
LIN {X 0,Y 172.3,Z 283.992,A -85,B 0,C 180,E1 -22860.001,E2 -22860.001} C_VEL
LIN {X 0,Y 171.766,Z 284.087,A -85,B 0,C 180,E1 -22864.694,E2 -22864.694} C_VEL
LIN {X 0,Y 171.833,Z 284.05,A -85,B 0,C 180,E1 -22869.417,E2 -22869.417} C_VEL
LIN {X 0,Y 171.549,Z 284.11,A -85,B 0,C 180,E1 -22874.23,E2 -22874.23} C_VEL
LIN {X 0,Y 171.474,Z 284.106,A -85,B 0,C 180,E1 -22879.501,E2 -22879.501} C_VEL
LIN {X 0,Y 171.396,Z 284.109,A -85,B 0,C 180,E1 -22885.57,E2 -22885.57} C_VEL
LIN {X 0,Y 171.401,Z 284.133,A -85,B 0,C 180,E1 -22890.567,E2 -22890.567} C_VEL
LIN {X 0,Y 171.388,Z 284.121,A -85,B 0,C 180,E1 -22895.037,E2 -22895.037} C_VEL
LIN {X 0,Y 171.339,Z 284.127,A -85,B 0,C 180,E1 -22898.803,E2 -22898.803} C_VEL
LIN {X 0,Y 171.314,Z 284.078,A -85,B 0,C 180,E1 -22904.22,E2 -22904.22} C_VEL
LIN {X 0,Y 171.327,Z 284.141,A -85,B 0,C 180,E1 -22908.982,E2 -22908.982} C_VEL
LIN {X 0,Y 171.408,Z 284.203,A -85,B 0,C 180,E1 -22914.274,E2 -22914.274} C_VEL
LIN {X 0,Y 171.625,Z 285.187,A -85,B 0,C 180,E1 -22914.861,E2 -22914.861} C_VEL
LIN {X 0,Y 173.121,Z 287.937,A -85,B 0,C 180,E1 -22915.472,E2 -22915.472} C_VEL
LIN {X 0,Y 174.158,Z 289.134,A -85,B 0,C 180,E1 -22915.818,E2 -22915.818} C_VEL
LIN {X 0,Y 183.037,Z 304.018,A -85,B 0,C 180,E1 -22918.786,E2 -22918.786} C_VEL
LIN {X 0,Y 190.781,Z 319.209,A -85,B 0,C 180,E1 -22921.172,E2 -22921.172} C_VEL
LIN {X 0,Y 193.439,Z 325.353,A -85,B 0,C 180,E1 -22921.973,E2 -22921.973} C_VEL
LIN {X 0,Y 191.716,Z 371.101,A -85,B 0,C 180,E1 -22923.697,E2 -22923.697} C_VEL
LIN {X 0,Y 190.981,Z 382.401,A -85,B 0,C 180,E1 -22924.455,E2 -22924.455} C_VEL
LIN {X 0,Y 189.658,Z 394.757,A -85,B 0,C 180,E1 -22925.655,E2 -22925.655} C_VEL
LIN {X 0,Y 187.86,Z 406.345,A -85,B 0,C 180,E1 -22927.163,E2 -22927.163} C_VEL
LIN {X 0,Y 185.797,Z 416.916,A -85,B 0,C 180,E1 -22928.941,E2 -22928.941} C_VEL
LIN {X 0,Y 183.38,Z 427.698,A -85,B 0,C 180,E1 -22931.28,E2 -22931.28} C_VEL
LIN {X 0,Y 180.662,Z 438.245,A -85,B 0,C 180,E1 -22934.2,E2 -22934.2} C_VEL
LIN {X 0,Y 178.447,Z 446.039,A -85,B 0,C 180,E1 -22936.913,E2 -22936.913} C_VEL
LIN {X 0,Y 176.119,Z 453.682,A -85,B 0,C 180,E1 -22940.237,E2 -22940.237} C_VEL
LIN {X 0,Y 174.05,Z 460.7,A -85,B 0,C 180,E1 -22944.207,E2 -22944.207} C_VEL
LIN {X 0,Y 172.702,Z 465.399,A -85,B 0,C 180,E1 -22947.669,E2 -22947.669} C_VEL
LIN {X 0,Y 171.751,Z 469.019,A -85,B 0,C 180,E1 -22951.173,E2 -22951.173} C_VEL
LIN {X 0,Y 171.375,Z 471.629,A -85,B 0,C 180,E1 -22954.705,E2 -22954.705} C_VEL
LIN {X 0,Y 171.371,Z 472.873,A -85,B 0,C 180,E1 -22957.068,E2 -22957.068} C_VEL
LIN {X 0,Y 171.653,Z 473.986,A -85,B 0,C 180,E1 -22960.69,E2 -22960.69} C_VEL
LIN {X 0,Y 172.312,Z 474.193,A -85,B 0,C 180,E1 -22964.166,E2 -22964.166} C_VEL
LIN {X 0,Y 173.051,Z 473.866,A -85,B 0,C 180,E1 -22966.517,E2 -22966.517} C_VEL
LIN {X 0,Y 174.017,Z 473.115,A -85,B 0,C 180,E1 -22968.851,E2 -22968.851} C_VEL
LIN {X 0,Y 176.619,Z 470.375,A -85,B 0,C 180,E1 -22973.449,E2 -22973.449} C_VEL
LIN {X 0,Y 179.081,Z 467.18,A -85,B 0,C 180,E1 -22976.828,E2 -22976.828} C_VEL
LIN {X 0,Y 182.072,Z 462.888,A -85,B 0,C 180,E1 -22980.12,E2 -22980.12} C_VEL
LIN {X 0,Y 185.686,Z 457.179,A -85,B 0,C 180,E1 -22983.41,E2 -22983.41} C_VEL
LIN {X 0,Y 189.458,Z 450.399,A -85,B 0,C 180,E1 -22986.408,E2 -22986.408} C_VEL
LIN {X 0,Y 193.859,Z 441.61,A -85,B 0,C 180,E1 -22989.378,E2 -22989.378} C_VEL
LIN {X 0,Y 197.918,Z 431.997,A -85,B 0,C 180,E1 -22991.931,E2 -22991.931} C_VEL
LIN {X 0,Y 201.37,Z 422.399,A -85,B 0,C 180,E1 -22993.92,E2 -22993.92} C_VEL
LIN {X 0,Y 204.754,Z 411.035,A -85,B 0,C 180,E1 -22995.767,E2 -22995.767} C_VEL
LIN {X 0,Y 207.475,Z 399.747,A -85,B 0,C 180,E1 -22997.171,E2 -22997.171} C_VEL
LIN {X 0,Y 209.662,Z 387.53,A -85,B 0,C 180,E1 -22998.303,E2 -22998.303} C_VEL
LIN {X 0,Y 210.819,Z 376.497,A -85,B 0,C 180,E1 -22999.086,E2 -22999.086} C_VEL
LIN {X 0,Y 211.827,Z 359.602,A -85,B 0,C 180,E1 -22999.788,E2 -22999.788} C_VEL
LIN {X 0,Y 212.534,Z 344.175,A -85,B 0,C 180,E1 -23000.332,E2 -23000.332} C_VEL
LIN {X 0,Y 205.964,Z 331.983,A -85,B 0,C 180,E1 -23002.949,E2 -23002.949} C_VEL
LIN {X 0,Y 199.07,Z 320.682,A -85,B 0,C 180,E1 -23005.974,E2 -23005.974} C_VEL
LIN {X 0,Y 193.976,Z 313.2,A -85,B 0,C 180,E1 -23008.45,E2 -23008.45} C_VEL
LIN {X 0,Y 190.796,Z 308.825,A -85,B 0,C 180,E1 -23010.129,E2 -23010.129} C_VEL
LIN {X 0,Y 187.942,Z 304.917,A -85,B 0,C 180,E1 -23011.752,E2 -23011.752} C_VEL
LIN {X 0,Y 185.191,Z 301.316,A -85,B 0,C 180,E1 -23013.432,E2 -23013.432} C_VEL
LIN {X 0,Y 184.13,Z 300.084,A -85,B 0,C 180,E1 -23014.106,E2 -23014.106} C_VEL
LIN {X 0,Y 181.655,Z 297.193,A -85,B 0,C 180,E1 -23015.769,E2 -23015.769} C_VEL
LIN {X 0,Y 180.475,Z 295.275,A -85,B 0,C 180,E1 -23016.66,E2 -23016.66} C_VEL
LIN {X 0,Y 177.749,Z 292.746,A -85,B 0,C 180,E1 -23018.699,E2 -23018.699} C_VEL
LIN {X 0,Y 176.186,Z 289.976,A -85,B 0,C 180,E1 -23020.106,E2 -23020.106} C_VEL
LIN {X 0,Y 173.09,Z 287.695,A -85,B 0,C 180,E1 -23022.879,E2 -23022.879} C_VEL
LIN {X 0,Y 171.678,Z 284.701,A -85,B 0,C 180,E1 -23024.872,E2 -23024.872} C_VEL
LIN {X 0,Y 171.623,Z 284.122,A -85,B 0,C 180,E1 -23026.38,E2 -23026.38} C_VEL
LIN {X 0,Y 171.842,Z 284.058,A -85,B 0,C 180,E1 -23030.584,E2 -23030.584} C_VEL
LIN {X 0,Y 171.776,Z 284.068,A -85,B 0,C 180,E1 -23035.306,E2 -23035.306} C_VEL
LIN {X 0,Y 172.307,Z 284.01,A -85,B 0,C 180,E1 -23039.999,E2 -23039.999} C_VEL
LIN {X 0,Y 171.783,Z 284.088,A -85,B 0,C 180,E1 -23044.693,E2 -23044.693} C_VEL
LIN {X 0,Y 171.84,Z 284.068,A -85,B 0,C 180,E1 -23049.415,E2 -23049.415} C_VEL
LIN {X 0,Y 171.564,Z 284.096,A -85,B 0,C 180,E1 -23054.228,E2 -23054.228} C_VEL
LIN {X 0,Y 171.609,Z 284.253,A -85,B 0,C 180,E1 -23058.814,E2 -23058.814} C_VEL
LIN {X 0,Y 173.063,Z 288.26,A -85,B 0,C 180,E1 -23063.324,E2 -23063.324} C_VEL
LIN {X 0,Y 179.415,Z 297.758,A -85,B 0,C 180,E1 -23069.237,E2 -23069.237} C_VEL
LIN {X 0,Y 184.486,Z 305.591,A -85,B 0,C 180,E1 -23072.874,E2 -23072.874} C_VEL
LIN {X 0,Y 188.759,Z 312.7,A -85,B 0,C 180,E1 -23075.554,E2 -23075.554} C_VEL
LIN {X 0,Y 192.917,Z 320.152,A -85,B 0,C 180,E1 -23077.918,E2 -23077.918} C_VEL
LIN {X 0,Y 196.339,Z 326.671,A -85,B 0,C 180,E1 -23079.716,E2 -23079.716} C_VEL
LIN {X 0,Y 201.871,Z 338.124,A -85,B 0,C 180,E1 -23082.407,E2 -23082.407} C_VEL
LIN {X 0,Y 206.907,Z 350.295,A -85,B 0,C 180,E1 -23084.695,E2 -23084.695} C_VEL
LIN {X 0,Y 208.697,Z 370.631,A -85,B 0,C 180,E1 -23086.251,E2 -23086.251} C_VEL
LIN {X 0,Y 209.835,Z 389.154,A -85,B 0,C 180,E1 -23087.472,E2 -23087.472} C_VEL
LIN {X 0,Y 208.408,Z 409.715,A -85,B 0,C 180,E1 -23088.162,E2 -23088.162} C_VEL
LIN {X 0,Y 206.331,Z 423.558,A -85,B 0,C 180,E1 -23088.901,E2 -23088.901} C_VEL
LIN {X 0,Y 203.784,Z 435.5,A -85,B 0,C 180,E1 -23089.873,E2 -23089.873} C_VEL
LIN {X 0,Y 200.513,Z 447.34,A -85,B 0,C 180,E1 -23091.206,E2 -23091.206} C_VEL
LIN {X 0,Y 196.189,Z 459.393,A -85,B 0,C 180,E1 -23092.964,E2 -23092.964} C_VEL
LIN {X 0,Y 193.739,Z 464.162,A -85,B 0,C 180,E1 -23093.697,E2 -23093.697} C_VEL
LIN {X 0,Y 188.063,Z 471.482,A -85,B 0,C 180,E1 -23094.771,E2 -23094.771} C_VEL
LIN {X 0,Y 182.235,Z 478.26,A -85,B 0,C 180,E1 -23096.09,E2 -23096.09} C_VEL
LIN {X 0,Y 179.591,Z 482.177,A -85,B 0,C 180,E1 -23097.207,E2 -23097.207} C_VEL
LIN {X 0,Y 174.795,Z 490.858,A -85,B 0,C 180,E1 -23100.492,E2 -23100.492} C_VEL
LIN {X 0,Y 171.522,Z 496.419,A -85,B 0,C 180,E1 -23103.21,E2 -23103.21} C_VEL
LIN {X 0,Y 167.941,Z 502.499,A -85,B 0,C 180,E1 -23107.022,E2 -23107.022} C_VEL
LIN {X 0,Y 165.149,Z 507.516,A -85,B 0,C 180,E1 -23111.387,E2 -23111.387} C_VEL
LIN {X 0,Y 163.578,Z 510.534,A -85,B 0,C 180,E1 -23115.061,E2 -23115.061} C_VEL
LIN {X 0,Y 162.74,Z 513.129,A -85,B 0,C 180,E1 -23120.052,E2 -23120.052} C_VEL
LIN {X 0,Y 162.884,Z 513.927,A -85,B 0,C 180,E1 -23122.925,E2 -23122.925} C_VEL
LIN {X 0,Y 163.584,Z 514.053,A -85,B 0,C 180,E1 -23127.537,E2 -23127.537} C_VEL
LIN {X 0,Y 163.825,Z 513.501,A -85,B 0,C 180,E1 -23129.999,E2 -23129.999} C_VEL
LIN {X 0,Y 163.557,Z 512.461,A -85,B 0,C 180,E1 -23132.462,E2 -23132.462} C_VEL
LIN {X 0,Y 163.151,Z 510.921,A -85,B 0,C 180,E1 -23134.941,E2 -23134.941} C_VEL
LIN {X 0,Y 162.854,Z 507.765,A -85,B 0,C 180,E1 -23138.686,E2 -23138.686} C_VEL
LIN {X 0,Y 163.099,Z 503.517,A -85,B 0,C 180,E1 -23142.441,E2 -23142.441} C_VEL
LIN {X 0,Y 164.219,Z 497.033,A -85,B 0,C 180,E1 -23146.789,E2 -23146.789} C_VEL
LIN {X 0,Y 165.917,Z 490.088,A -85,B 0,C 180,E1 -23150.409,E2 -23150.409} C_VEL
LIN {X 0,Y 168.022,Z 482.87,A -85,B 0,C 180,E1 -23153.411,E2 -23153.411} C_VEL
LIN {X 0,Y 170.582,Z 474.289,A -85,B 0,C 180,E1 -23156.287,E2 -23156.287} C_VEL
LIN {X 0,Y 173.2,Z 464.872,A -85,B 0,C 180,E1 -23158.805,E2 -23158.805} C_VEL
LIN {X 0,Y 175.666,Z 456.12,A -85,B 0,C 180,E1 -23160.668,E2 -23160.668} C_VEL
LIN {X 0,Y 178.3,Z 445.374,A -85,B 0,C 180,E1 -23162.481,E2 -23162.481} C_VEL
LIN {X 0,Y 180.639,Z 433.55,A -85,B 0,C 180,E1 -23164.004,E2 -23164.004} C_VEL
LIN {X 0,Y 182.563,Z 420.878,A -85,B 0,C 180,E1 -23165.185,E2 -23165.185} C_VEL
LIN {X 0,Y 183.713,Z 408.329,A -85,B 0,C 180,E1 -23165.98,E2 -23165.98} C_VEL
LIN {X 0,Y 184.879,Z 383.442,A -85,B 0,C 180,E1 -23166.92,E2 -23166.92} C_VEL
LIN {X 0,Y 182.741,Z 346.763,A -85,B 0,C 180,E1 -23169.042,E2 -23169.042} C_VEL
LIN {X 0,Y 181.169,Z 327.172,A -85,B 0,C 180,E1 -23170.314,E2 -23170.314} C_VEL
LIN {X 0,Y 174.935,Z 311.395,A -85,B 0,C 180,E1 -23172.597,E2 -23172.597} C_VEL
LIN {X 0,Y 169.197,Z 299.746,A -85,B 0,C 180,E1 -23174.763,E2 -23174.763} C_VEL
LIN {X 0,Y 167.415,Z 295.791,A -85,B 0,C 180,E1 -23175.658,E2 -23175.658} C_VEL
LIN {X 0,Y 165,Z 287.343,A -85,B 0,C 180,E1 -23180.29,E2 -23180.29} C_VEL
LIN {X 0,Y 164.339,Z 285.084,A -85,B 0,C 180,E1 -23181.775,E2 -23181.775} C_VEL
LIN {X 0,Y 164.312,Z 284.995,A -85,B 0,C 180,E1 -23186.218,E2 -23186.218} C_VEL
LIN {X 0,Y 164.36,Z 284.99,A -85,B 0,C 180,E1 -23189.129,E2 -23189.129} C_VEL
LIN {X 0,Y 164.387,Z 284.986,A -85,B 0,C 180,E1 -23194.69,E2 -23194.69} C_VEL
LIN {X 0,Y 164.41,Z 284.99,A -85,B 0,C 180,E1 -23200.117,E2 -23200.117} C_VEL
LIN {X 0,Y 164.476,Z 284.994,A -85,B 0,C 180,E1 -23205.145,E2 -23205.145} C_VEL
LIN {X 0,Y 164.756,Z 284.932,A -85,B 0,C 180,E1 -23210.176,E2 -23210.176} C_VEL
LIN {X 0,Y 164.811,Z 284.941,A -85,B 0,C 180,E1 -23212.651,E2 -23212.651} C_VEL
LIN {X 0,Y 165.264,Z 284.867,A -85,B 0,C 180,E1 -23220.001,E2 -23220.001} C_VEL
LIN {X 0,Y 164.807,Z 284.926,A -85,B 0,C 180,E1 -23227.351,E2 -23227.351} C_VEL
LIN {X 0,Y 164.695,Z 284.954,A -85,B 0,C 180,E1 -23231.057,E2 -23231.057} C_VEL
LIN {X 0,Y 164.43,Z 284.97,A -85,B 0,C 180,E1 -23237.41,E2 -23237.41} C_VEL
LIN {X 0,Y 164.414,Z 284.991,A -85,B 0,C 180,E1 -23239.997,E2 -23239.997} C_VEL
LIN {X 0,Y 164.33,Z 284.987,A -85,B 0,C 180,E1 -23246.093,E2 -23246.093} C_VEL
LIN {X 0,Y 164.339,Z 285.007,A -85,B 0,C 180,E1 -23251.211,E2 -23251.211} C_VEL
LIN {X 0,Y 164.276,Z 285.023,A -85,B 0,C 180,E1 -23256.795,E2 -23256.795} C_VEL
LIN {X 0,Y 164.282,Z 284.977,A -85,B 0,C 180,E1 -23259.92,E2 -23259.92} C_VEL
LIN {X 0,Y 164.277,Z 284.947,A -85,B 0,C 180,E1 -23263.344,E2 -23263.344} C_VEL
LIN {X 0,Y 164.257,Z 284.993,A -85,B 0,C 180,E1 -23266.8,E2 -23266.8} C_VEL
LIN {X 0,Y 164.36,Z 285.168,A -85,B 0,C 180,E1 -23272.267,E2 -23272.267} C_VEL
LIN {X 0,Y 164.553,Z 286.07,A -85,B 0,C 180,E1 -23272.781,E2 -23272.781} C_VEL
LIN {X 0,Y 166.037,Z 288.764,A -85,B 0,C 180,E1 -23273.454,E2 -23273.454} C_VEL
LIN {X 0,Y 167.354,Z 290.432,A -85,B 0,C 180,E1 -23273.95,E2 -23273.95} C_VEL
LIN {X 0,Y 169.56,Z 293.727,A -85,B 0,C 180,E1 -23274.781,E2 -23274.781} C_VEL
LIN {X 0,Y 177.917,Z 307.741,A -85,B 0,C 180,E1 -23277.742,E2 -23277.742} C_VEL
LIN {X 0,Y 185.002,Z 321.803,A -85,B 0,C 180,E1 -23280.07,E2 -23280.07} C_VEL
LIN {X 0,Y 187.447,Z 327.188,A -85,B 0,C 180,E1 -23280.843,E2 -23280.843} C_VEL
LIN {X 0,Y 185.716,Z 371.748,A -85,B 0,C 180,E1 -23282.573,E2 -23282.573} C_VEL
LIN {X 0,Y 184.959,Z 382.882,A -85,B 0,C 180,E1 -23283.332,E2 -23283.332} C_VEL
LIN {X 0,Y 183.473,Z 395.89,A -85,B 0,C 180,E1 -23284.627,E2 -23284.627} C_VEL
LIN {X 0,Y 181.421,Z 408.283,A -85,B 0,C 180,E1 -23286.304,E2 -23286.304} C_VEL
LIN {X 0,Y 178.977,Z 419.876,A -85,B 0,C 180,E1 -23288.401,E2 -23288.401} C_VEL
LIN {X 0,Y 176.488,Z 430.257,A -85,B 0,C 180,E1 -23290.822,E2 -23290.822} C_VEL
LIN {X 0,Y 173.914,Z 439.642,A -85,B 0,C 180,E1 -23293.57,E2 -23293.57} C_VEL
LIN {X 0,Y 171.131,Z 448.691,A -85,B 0,C 180,E1 -23296.947,E2 -23296.947} C_VEL
LIN {X 0,Y 168.8,Z 455.984,A -85,B 0,C 180,E1 -23300.415,E2 -23300.415} C_VEL
LIN {X 0,Y 167.045,Z 461.828,A -85,B 0,C 180,E1 -23303.964,E2 -23303.964} C_VEL
LIN {X 0,Y 165.646,Z 466.469,A -85,B 0,C 180,E1 -23307.569,E2 -23307.569} C_VEL
LIN {X 0,Y 164.688,Z 470.034,A -85,B 0,C 180,E1 -23311.224,E2 -23311.224} C_VEL
LIN {X 0,Y 164.33,Z 472.593,A -85,B 0,C 180,E1 -23314.908,E2 -23314.908} C_VEL
LIN {X 0,Y 164.337,Z 473.809,A -85,B 0,C 180,E1 -23317.372,E2 -23317.372} C_VEL
LIN {X 0,Y 164.862,Z 475.004,A -85,B 0,C 180,E1 -23322.308,E2 -23322.308} C_VEL
LIN {X 0,Y 166.228,Z 474.68,A -85,B 0,C 180,E1 -23327.215,E2 -23327.215} C_VEL
LIN {X 0,Y 168.552,Z 472.692,A -85,B 0,C 180,E1 -23332.041,E2 -23332.041} C_VEL
LIN {X 0,Y 170.319,Z 470.806,A -85,B 0,C 180,E1 -23334.795,E2 -23334.795} C_VEL
LIN {X 0,Y 173.724,Z 466.509,A -85,B 0,C 180,E1 -23339.043,E2 -23339.043} C_VEL
LIN {X 0,Y 177.091,Z 461.759,A -85,B 0,C 180,E1 -23342.396,E2 -23342.396} C_VEL
LIN {X 0,Y 180.924,Z 455.715,A -85,B 0,C 180,E1 -23345.639,E2 -23345.639} C_VEL
LIN {X 0,Y 185.241,Z 448.123,A -85,B 0,C 180,E1 -23348.756,E2 -23348.756} C_VEL
LIN {X 0,Y 189.154,Z 440.278,A -85,B 0,C 180,E1 -23351.262,E2 -23351.262} C_VEL
LIN {X 0,Y 193.232,Z 430.643,A -85,B 0,C 180,E1 -23353.713,E2 -23353.713} C_VEL
LIN {X 0,Y 197.153,Z 419.857,A -85,B 0,C 180,E1 -23355.84,E2 -23355.84} C_VEL
LIN {X 0,Y 200.266,Z 409.244,A -85,B 0,C 180,E1 -23357.473,E2 -23357.473} C_VEL
LIN {X 0,Y 202.966,Z 397.832,A -85,B 0,C 180,E1 -23358.805,E2 -23358.805} C_VEL
LIN {X 0,Y 204.867,Z 386.487,A -85,B 0,C 180,E1 -23359.828,E2 -23359.828} C_VEL
LIN {X 0,Y 205.974,Z 376.162,A -85,B 0,C 180,E1 -23360.525,E2 -23360.525} C_VEL
LIN {X 0,Y 207.048,Z 358.485,A -85,B 0,C 180,E1 -23361.242,E2 -23361.242} C_VEL
LIN {X 0,Y 207.521,Z 346.813,A -85,B 0,C 180,E1 -23361.689,E2 -23361.689} C_VEL
LIN {X 0,Y 201.627,Z 335.885,A -85,B 0,C 180,E1 -23364.191,E2 -23364.191} C_VEL
LIN {X 0,Y 195.489,Z 325.646,A -85,B 0,C 180,E1 -23367.059,E2 -23367.059} C_VEL
LIN {X 0,Y 190.627,Z 318.377,A -85,B 0,C 180,E1 -23369.567,E2 -23369.567} C_VEL
LIN {X 0,Y 187.872,Z 314.455,A -85,B 0,C 180,E1 -23371.111,E2 -23371.111} C_VEL
LIN {X 0,Y 185.144,Z 310.716,A -85,B 0,C 180,E1 -23372.748,E2 -23372.748} C_VEL
LIN {X 0,Y 182.111,Z 306.621,A -85,B 0,C 180,E1 -23374.727,E2 -23374.727} C_VEL
LIN {X 0,Y 179.302,Z 303.209,A -85,B 0,C 180,E1 -23376.71,E2 -23376.71} C_VEL
LIN {X 0,Y 178.397,Z 301.7,A -85,B 0,C 180,E1 -23377.43,E2 -23377.43} C_VEL
LIN {X 0,Y 175.783,Z 299.096,A -85,B 0,C 180,E1 -23379.494,E2 -23379.494} C_VEL
LIN {X 0,Y 174.298,Z 296.577,A -85,B 0,C 180,E1 -23380.885,E2 -23380.885} C_VEL
LIN {X 0,Y 171.413,Z 294.217,A -85,B 0,C 180,E1 -23383.627,E2 -23383.627} C_VEL
LIN {X 0,Y 169.797,Z 291.179,A -85,B 0,C 180,E1 -23385.62,E2 -23385.62} C_VEL
LIN {X 0,Y 166.691,Z 289.014,A -85,B 0,C 180,E1 -23389.733,E2 -23389.733} C_VEL
LIN {X 0,Y 165.129,Z 286.35,A -85,B 0,C 180,E1 -23392.894,E2 -23392.894} C_VEL
LIN {X 0,Y 164.824,Z 285.435,A -85,B 0,C 180,E1 -23394.494,E2 -23394.494} C_VEL
LIN {X 0,Y 165.018,Z 284.953,A -85,B 0,C 180,E1 -23397.559,E2 -23397.559} C_VEL
LIN {X 0,Y 165.271,Z 284.886,A -85,B 0,C 180,E1 -23399.999,E2 -23399.999} C_VEL
LIN {X 0,Y 164.817,Z 284.96,A -85,B 0,C 180,E1 -23407.349,E2 -23407.349} C_VEL
LIN {X 0,Y 164.748,Z 285.234,A -85,B 0,C 180,E1 -23411.142,E2 -23411.142} C_VEL
LIN {X 0,Y 164.9,Z 286.468,A -85,B 0,C 180,E1 -23413.086,E2 -23413.086} C_VEL
LIN {X 0,Y 166.404,Z 289.009,A -85,B 0,C 180,E1 -23416.248,E2 -23416.248} C_VEL
LIN {X 0,Y 168.101,Z 290.548,A -85,B 0,C 180,E1 -23418.747,E2 -23418.747} C_VEL
LIN {X 0,Y 171.542,Z 295.328,A -85,B 0,C 180,E1 -23422.985,E2 -23422.985} C_VEL
LIN {X 0,Y 177.287,Z 304.088,A -85,B 0,C 180,E1 -23428.405,E2 -23428.405} C_VEL
LIN {X 0,Y 181.837,Z 311.328,A -85,B 0,C 180,E1 -23431.857,E2 -23431.857} C_VEL
LIN {X 0,Y 185.877,Z 318.339,A -85,B 0,C 180,E1 -23434.551,E2 -23434.551} C_VEL
LIN {X 0,Y 189.924,Z 325.792,A -85,B 0,C 180,E1 -23436.984,E2 -23436.984} C_VEL
LIN {X 0,Y 194.501,Z 334.97,A -85,B 0,C 180,E1 -23439.497,E2 -23439.497} C_VEL
LIN {X 0,Y 199.3,Z 345.757,A -85,B 0,C 180,E1 -23441.933,E2 -23441.933} C_VEL
LIN {X 0,Y 202.405,Z 353.635,A -85,B 0,C 180,E1 -23443.431,E2 -23443.431} C_VEL
LIN {X 0,Y 204.079,Z 375.121,A -85,B 0,C 180,E1 -23445.094,E2 -23445.094} C_VEL
LIN {X 0,Y 204.832,Z 390.378,A -85,B 0,C 180,E1 -23446.098,E2 -23446.098} C_VEL
LIN {X 0,Y 203.361,Z 409.865,A -85,B 0,C 180,E1 -23446.775,E2 -23446.775} C_VEL
LIN {X 0,Y 201.285,Z 423.029,A -85,B 0,C 180,E1 -23447.497,E2 -23447.497} C_VEL
LIN {X 0,Y 198.671,Z 434.669,A -85,B 0,C 180,E1 -23448.449,E2 -23448.449} C_VEL
LIN {X 0,Y 195.032,Z 447.29,A -85,B 0,C 180,E1 -23449.9,E2 -23449.9} C_VEL
LIN {X 0,Y 190.823,Z 458.563,A -85,B 0,C 180,E1 -23451.574,E2 -23451.574} C_VEL
LIN {X 0,Y 186.345,Z 468.749,A -85,B 0,C 180,E1 -23453.558,E2 -23453.558} C_VEL
LIN {X 0,Y 181.784,Z 477.964,A -85,B 0,C 180,E1 -23455.903,E2 -23455.903} C_VEL
LIN {X 0,Y 179.591,Z 482.177,A -85,B 0,C 180,E1 -23457.207,E2 -23457.207} C_VEL
LIN {X 0,Y 176.964,Z 485.954,A -85,B 0,C 180,E1 -23458.424,E2 -23458.424} C_VEL
LIN {X 0,Y 171.131,Z 491.533,A -85,B 0,C 180,E1 -23460.34,E2 -23460.34} C_VEL
LIN {X 0,Y 165.448,Z 496.456,A -85,B 0,C 180,E1 -23462.529,E2 -23462.529} C_VEL
LIN {X 0,Y 163.113,Z 499.152,A -85,B 0,C 180,E1 -23464.146,E2 -23464.146} C_VEL
LIN {X 0,Y 159.864,Z 504.271,A -85,B 0,C 180,E1 -23468.057,E2 -23468.057} C_VEL
LIN {X 0,Y 157.746,Z 507.91,A -85,B 0,C 180,E1 -23471.827,E2 -23471.827} C_VEL
LIN {X 0,Y 156.027,Z 511.233,A -85,B 0,C 180,E1 -23476.984,E2 -23476.984} C_VEL
LIN {X 0,Y 155.765,Z 513.023,A -85,B 0,C 180,E1 -23482.22,E2 -23482.22} C_VEL
LIN {X 0,Y 156.493,Z 513.167,A -85,B 0,C 180,E1 -23487.425,E2 -23487.425} C_VEL
LIN {X 0,Y 156.776,Z 512.603,A -85,B 0,C 180,E1 -23489.999,E2 -23489.999} C_VEL
LIN {X 0,Y 156.463,Z 511.532,A -85,B 0,C 180,E1 -23492.573,E2 -23492.573} C_VEL
LIN {X 0,Y 155.88,Z 508.329,A -85,B 0,C 180,E1 -23497.303,E2 -23497.303} C_VEL
LIN {X 0,Y 155.937,Z 503.998,A -85,B 0,C 180,E1 -23501.7,E2 -23501.7} C_VEL
LIN {X 0,Y 156.692,Z 498.92,A -85,B 0,C 180,E1 -23505.61,E2 -23505.61} C_VEL
LIN {X 0,Y 158.135,Z 492.546,A -85,B 0,C 180,E1 -23509.469,E2 -23509.469} C_VEL
LIN {X 0,Y 160.569,Z 484.672,A -85,B 0,C 180,E1 -23513.197,E2 -23513.197} C_VEL
LIN {X 0,Y 163.057,Z 476.61,A -85,B 0,C 180,E1 -23516.216,E2 -23516.216} C_VEL
LIN {X 0,Y 165.672,Z 467.87,A -85,B 0,C 180,E1 -23518.85,E2 -23518.85} C_VEL
LIN {X 0,Y 168.868,Z 457.244,A -85,B 0,C 180,E1 -23521.346,E2 -23521.346} C_VEL
LIN {X 0,Y 171.921,Z 445.39,A -85,B 0,C 180,E1 -23523.493,E2 -23523.493} C_VEL
LIN {X 0,Y 174.351,Z 433.822,A -85,B 0,C 180,E1 -23525.056,E2 -23525.056} C_VEL
LIN {X 0,Y 176.458,Z 420.773,A -85,B 0,C 180,E1 -23526.328,E2 -23526.328} C_VEL
LIN {X 0,Y 177.738,Z 407.627,A -85,B 0,C 180,E1 -23527.2,E2 -23527.2} C_VEL
LIN {X 0,Y 178.928,Z 384.685,A -85,B 0,C 180,E1 -23528.079,E2 -23528.079} C_VEL
LIN {X 0,Y 177.023,Z 348.979,A -85,B 0,C 180,E1 -23530.215,E2 -23530.215} C_VEL
LIN {X 0,Y 175.574,Z 329.676,A -85,B 0,C 180,E1 -23531.514,E2 -23531.514} C_VEL
LIN {X 0,Y 169.772,Z 314.778,A -85,B 0,C 180,E1 -23533.793,E2 -23533.793} C_VEL
LIN {X 0,Y 164.57,Z 304.005,A -85,B 0,C 180,E1 -23535.897,E2 -23535.897} C_VEL
LIN {X 0,Y 159.93,Z 294.858,A -85,B 0,C 180,E1 -23538.026,E2 -23538.026} C_VEL
LIN {X 0,Y 158.131,Z 288.864,A -85,B 0,C 180,E1 -23541.522,E2 -23541.522} C_VEL
LIN {X 0,Y 157.261,Z 285.955,A -85,B 0,C 180,E1 -23543.551,E2 -23543.551} C_VEL
LIN {X 0,Y 157.274,Z 285.865,A -85,B 0,C 180,E1 -23548.103,E2 -23548.103} C_VEL
LIN {X 0,Y 157.303,Z 285.872,A -85,B 0,C 180,E1 -23553.463,E2 -23553.463} C_VEL
LIN {X 0,Y 157.353,Z 285.873,A -85,B 0,C 180,E1 -23559.702,E2 -23559.702} C_VEL
LIN {X 0,Y 157.408,Z 285.866,A -85,B 0,C 180,E1 -23564.462,E2 -23564.462} C_VEL
LIN {X 0,Y 157.679,Z 285.813,A -85,B 0,C 180,E1 -23569.731,E2 -23569.731} C_VEL
LIN {X 0,Y 157.75,Z 285.815,A -85,B 0,C 180,E1 -23572.32,E2 -23572.32} C_VEL
LIN {X 0,Y 158.227,Z 285.742,A -85,B 0,C 180,E1 -23580.001,E2 -23580.001} C_VEL
LIN {X 0,Y 157.746,Z 285.802,A -85,B 0,C 180,E1 -23587.682,E2 -23587.682} C_VEL
LIN {X 0,Y 157.625,Z 285.835,A -85,B 0,C 180,E1 -23591.226,E2 -23591.226} C_VEL
LIN {X 0,Y 157.409,Z 285.855,A -85,B 0,C 180,E1 -23595.539,E2 -23595.539} C_VEL
LIN {X 0,Y 157.299,Z 285.887,A -85,B 0,C 180,E1 -23600.943,E2 -23600.943} C_VEL
LIN {X 0,Y 157.262,Z 285.868,A -85,B 0,C 180,E1 -23606.651,E2 -23606.651} C_VEL
LIN {X 0,Y 157.256,Z 285.876,A -85,B 0,C 180,E1 -23612.433,E2 -23612.433} C_VEL
LIN {X 0,Y 157.254,Z 285.895,A -85,B 0,C 180,E1 -23616.446,E2 -23616.446} C_VEL
LIN {X 0,Y 157.185,Z 285.831,A -85,B 0,C 180,E1 -23622.12,E2 -23622.12} C_VEL
LIN {X 0,Y 157.187,Z 285.897,A -85,B 0,C 180,E1 -23627.884,E2 -23627.884} C_VEL
LIN {X 0,Y 157.289,Z 286.18,A -85,B 0,C 180,E1 -23630.046,E2 -23630.046} C_VEL
LIN {X 0,Y 157.66,Z 287.463,A -85,B 0,C 180,E1 -23630.571,E2 -23630.571} C_VEL
LIN {X 0,Y 159.148,Z 289.857,A -85,B 0,C 180,E1 -23631.266,E2 -23631.266} C_VEL
LIN {X 0,Y 160.386,Z 291.288,A -85,B 0,C 180,E1 -23631.778,E2 -23631.778} C_VEL
LIN {X 0,Y 162.652,Z 294.673,A -85,B 0,C 180,E1 -23632.729,E2 -23632.729} C_VEL
LIN {X 0,Y 168.411,Z 303.902,A -85,B 0,C 180,E1 -23635.008,E2 -23635.008} C_VEL
LIN {X 0,Y 174.804,Z 315.104,A -85,B 0,C 180,E1 -23637.332,E2 -23637.332} C_VEL
LIN {X 0,Y 181.534,Z 329.255,A -85,B 0,C 180,E1 -23639.65,E2 -23639.65} C_VEL
LIN {X 0,Y 179.664,Z 373.48,A -85,B 0,C 180,E1 -23641.43,E2 -23641.43} C_VEL
LIN {X 0,Y 178.848,Z 384.831,A -85,B 0,C 180,E1 -23642.265,E2 -23642.265} C_VEL
LIN {X 0,Y 177.223,Z 398.101,A -85,B 0,C 180,E1 -23643.664,E2 -23643.664} C_VEL
LIN {X 0,Y 175.02,Z 410.125,A -85,B 0,C 180,E1 -23645.381,E2 -23645.381} C_VEL
LIN {X 0,Y 172.48,Z 421.512,A -85,B 0,C 180,E1 -23647.544,E2 -23647.544} C_VEL
LIN {X 0,Y 169.882,Z 431.757,A -85,B 0,C 180,E1 -23650.045,E2 -23650.045} C_VEL
LIN {X 0,Y 167.187,Z 441.01,A -85,B 0,C 180,E1 -23652.888,E2 -23652.888} C_VEL
LIN {X 0,Y 164.276,Z 449.957,A -85,B 0,C 180,E1 -23656.392,E2 -23656.392} C_VEL
LIN {X 0,Y 161.855,Z 457.177,A -85,B 0,C 180,E1 -23659.999,E2 -23659.999} C_VEL
LIN {X 0,Y 160.044,Z 462.954,A -85,B 0,C 180,E1 -23663.698,E2 -23663.698} C_VEL
LIN {X 0,Y 158.592,Z 467.538,A -85,B 0,C 180,E1 -23667.461,E2 -23667.461} C_VEL
LIN {X 0,Y 157.599,Z 471.052,A -85,B 0,C 180,E1 -23671.279,E2 -23671.279} C_VEL
LIN {X 0,Y 157.287,Z 473.555,A -85,B 0,C 180,E1 -23675.128,E2 -23675.128} C_VEL
LIN {X 0,Y 157.31,Z 474.732,A -85,B 0,C 180,E1 -23677.703,E2 -23677.703} C_VEL
LIN {X 0,Y 157.91,Z 475.873,A -85,B 0,C 180,E1 -23682.859,E2 -23682.859} C_VEL
LIN {X 0,Y 158.526,Z 475.882,A -85,B 0,C 180,E1 -23685.427,E2 -23685.427} C_VEL
LIN {X 0,Y 159.437,Z 475.48,A -85,B 0,C 180,E1 -23687.973,E2 -23687.973} C_VEL
LIN {X 0,Y 161.963,Z 473.436,A -85,B 0,C 180,E1 -23692.988,E2 -23692.988} C_VEL
LIN {X 0,Y 163.734,Z 471.655,A -85,B 0,C 180,E1 -23695.657,E2 -23695.657} C_VEL
LIN {X 0,Y 166.44,Z 468.511,A -85,B 0,C 180,E1 -23699.052,E2 -23699.052} C_VEL
LIN {X 0,Y 169.839,Z 464.102,A -85,B 0,C 180,E1 -23702.544,E2 -23702.544} C_VEL
LIN {X 0,Y 174.061,Z 457.957,A -85,B 0,C 180,E1 -23706.143,E2 -23706.143} C_VEL
LIN {X 0,Y 178.911,Z 449.93,A -85,B 0,C 180,E1 -23709.668,E2 -23709.668} C_VEL
LIN {X 0,Y 182.998,Z 442.316,A -85,B 0,C 180,E1 -23712.228,E2 -23712.228} C_VEL
LIN {X 0,Y 187.464,Z 432.413,A -85,B 0,C 180,E1 -23714.862,E2 -23714.862} C_VEL
LIN {X 0,Y 191.747,Z 421.208,A -85,B 0,C 180,E1 -23717.143,E2 -23717.143} C_VEL
LIN {X 0,Y 195.004,Z 410.762,A -85,B 0,C 180,E1 -23718.793,E2 -23718.793} C_VEL
LIN {X 0,Y 198.011,Z 398.614,A -85,B 0,C 180,E1 -23720.237,E2 -23720.237} C_VEL
LIN {X 0,Y 200.018,Z 386.998,A -85,B 0,C 180,E1 -23721.296,E2 -23721.296} C_VEL
LIN {X 0,Y 201.277,Z 375.746,A -85,B 0,C 180,E1 -23722.036,E2 -23722.036} C_VEL
LIN {X 0,Y 202.515,Z 355.188,A -85,B 0,C 180,E1 -23722.845,E2 -23722.845} C_VEL
LIN {X 0,Y 202.711,Z 349.806,A -85,B 0,C 180,E1 -23723.068,E2 -23723.068} C_VEL
LIN {X 0,Y 197.943,Z 340.803,A -85,B 0,C 180,E1 -23725.228,E2 -23725.228} C_VEL
LIN {X 0,Y 192.051,Z 330.699,A -85,B 0,C 180,E1 -23728.15,E2 -23728.15} C_VEL
LIN {X 0,Y 187.863,Z 324.265,A -85,B 0,C 180,E1 -23730.434,E2 -23730.434} C_VEL
LIN {X 0,Y 184.436,Z 319.242,A -85,B 0,C 180,E1 -23732.481,E2 -23732.481} C_VEL
LIN {X 0,Y 181.934,Z 315.883,A -85,B 0,C 180,E1 -23734.087,E2 -23734.087} C_VEL
LIN {X 0,Y 179.601,Z 312.641,A -85,B 0,C 180,E1 -23735.714,E2 -23735.714} C_VEL
LIN {X 0,Y 176.794,Z 308.838,A -85,B 0,C 180,E1 -23737.85,E2 -23737.85} C_VEL
LIN {X 0,Y 175.399,Z 307.335,A -85,B 0,C 180,E1 -23738.966,E2 -23738.966} C_VEL
LIN {X 0,Y 172.898,Z 303.838,A -85,B 0,C 180,E1 -23741.234,E2 -23741.234} C_VEL
LIN {X 0,Y 172.107,Z 302.917,A -85,B 0,C 180,E1 -23741.992,E2 -23741.992} C_VEL
LIN {X 0,Y 169.623,Z 300.517,A -85,B 0,C 180,E1 -23744.559,E2 -23744.559} C_VEL
LIN {X 0,Y 168.183,Z 297.829,A -85,B 0,C 180,E1 -23746.443,E2 -23746.443} C_VEL
LIN {X 0,Y 165.491,Z 295.868,A -85,B 0,C 180,E1 -23750.219,E2 -23750.219} C_VEL
LIN {X 0,Y 163.561,Z 292.51,A -85,B 0,C 180,E1 -23754.451,E2 -23754.451} C_VEL
LIN {X 0,Y 162.057,Z 291.22,A -85,B 0,C 180,E1 -23759.999,E2 -23759.999} C_VEL
LIN {X 0,Y 162.854,Z 291.893,A -85,B 0,C 180,E1 -23769.94,E2 -23769.94} C_VEL
LIN {X 0,Y 163.54,Z 292.74,A -85,B 0,C 180,E1 -23771.963,E2 -23771.963} C_VEL
LIN {X 0,Y 165.031,Z 295.68,A -85,B 0,C 180,E1 -23775.436,E2 -23775.436} C_VEL
LIN {X 0,Y 166.819,Z 297.457,A -85,B 0,C 180,E1 -23778.265,E2 -23778.265} C_VEL
LIN {X 0,Y 169.745,Z 301.676,A -85,B 0,C 180,E1 -23782.077,E2 -23782.077} C_VEL
LIN {X 0,Y 175.05,Z 310.101,A -85,B 0,C 180,E1 -23787.416,E2 -23787.416} C_VEL
LIN {X 0,Y 179.527,Z 317.586,A -85,B 0,C 180,E1 -23791.023,E2 -23791.023} C_VEL
LIN {X 0,Y 183.146,Z 324.131,A -85,B 0,C 180,E1 -23793.578,E2 -23793.578} C_VEL
LIN {X 0,Y 187.106,Z 331.758,A -85,B 0,C 180,E1 -23796.1,E2 -23796.1} C_VEL
LIN {X 0,Y 192.256,Z 342.646,A -85,B 0,C 180,E1 -23799.069,E2 -23799.069} C_VEL
LIN {X 0,Y 197.067,Z 354.27,A -85,B 0,C 180,E1 -23801.617,E2 -23801.617} C_VEL
LIN {X 0,Y 197.948,Z 357.049,A -85,B 0,C 180,E1 -23802.092,E2 -23802.092} C_VEL
LIN {X 0,Y 199.498,Z 379.259,A -85,B 0,C 180,E1 -23803.85,E2 -23803.85} C_VEL
LIN {X 0,Y 199.963,Z 391.647,A -85,B 0,C 180,E1 -23804.662,E2 -23804.662} C_VEL
LIN {X 0,Y 198.481,Z 409.756,A -85,B 0,C 180,E1 -23805.311,E2 -23805.311} C_VEL
LIN {X 0,Y 196.559,Z 421.489,A -85,B 0,C 180,E1 -23805.958,E2 -23805.958} C_VEL
LIN {X 0,Y 193.726,Z 433.844,A -85,B 0,C 180,E1 -23806.962,E2 -23806.962} C_VEL
LIN {X 0,Y 190.174,Z 445.663,A -85,B 0,C 180,E1 -23808.302,E2 -23808.302} C_VEL
LIN {X 0,Y 185.817,Z 457.073,A -85,B 0,C 180,E1 -23809.986,E2 -23809.986} C_VEL
LIN {X 0,Y 181.191,Z 467.396,A -85,B 0,C 180,E1 -23811.993,E2 -23811.993} C_VEL
LIN {X 0,Y 175.943,Z 477.525,A -85,B 0,C 180,E1 -23814.606,E2 -23814.606} C_VEL
LIN {X 0,Y 170.932,Z 486.491,A -85,B 0,C 180,E1 -23817.689,E2 -23817.689} C_VEL
LIN {X 0,Y 166.509,Z 493.742,A -85,B 0,C 180,E1 -23820.961,E2 -23820.961} C_VEL
LIN {X 0,Y 163.113,Z 499.152,A -85,B 0,C 180,E1 -23824.146,E2 -23824.146} C_VEL
LIN {X 0,Y 160.896,Z 501.701,A -85,B 0,C 180,E1 -23825.864,E2 -23825.864} C_VEL
LIN {X 0,Y 155.833,Z 505.173,A -85,B 0,C 180,E1 -23828.691,E2 -23828.691} C_VEL
LIN {X 0,Y 151.195,Z 507.847,A -85,B 0,C 180,E1 -23831.81,E2 -23831.81} C_VEL
LIN {X 0,Y 149.702,Z 509.144,A -85,B 0,C 180,E1 -23833.931,E2 -23833.931} C_VEL
LIN {X 0,Y 148.689,Z 511.509,A -85,B 0,C 180,E1 -23839.101,E2 -23839.101} C_VEL
LIN {X 0,Y 148.765,Z 512.293,A -85,B 0,C 180,E1 -23842.787,E2 -23842.787} C_VEL
LIN {X 0,Y 149.404,Z 512.283,A -85,B 0,C 180,E1 -23847.303,E2 -23847.303} C_VEL
LIN {X 0,Y 149.725,Z 511.704,A -85,B 0,C 180,E1 -23849.999,E2 -23849.999} C_VEL
LIN {X 0,Y 149.37,Z 510.594,A -85,B 0,C 180,E1 -23852.696,E2 -23852.696} C_VEL
LIN {X 0,Y 148.8,Z 507.605,A -85,B 0,C 180,E1 -23857.319,E2 -23857.319} C_VEL
LIN {X 0,Y 148.923,Z 502.954,A -85,B 0,C 180,E1 -23862.26,E2 -23862.26} C_VEL
LIN {X 0,Y 149.786,Z 497.826,A -85,B 0,C 180,E1 -23866.349,E2 -23866.349} C_VEL
LIN {X 0,Y 151.406,Z 491.402,A -85,B 0,C 180,E1 -23870.372,E2 -23870.372} C_VEL
LIN {X 0,Y 153.996,Z 483.429,A -85,B 0,C 180,E1 -23874.249,E2 -23874.249} C_VEL
LIN {X 0,Y 156.687,Z 475.298,A -85,B 0,C 180,E1 -23877.369,E2 -23877.369} C_VEL
LIN {X 0,Y 159.788,Z 465.375,A -85,B 0,C 180,E1 -23880.383,E2 -23880.383} C_VEL
LIN {X 0,Y 162.76,Z 455.709,A -85,B 0,C 180,E1 -23882.665,E2 -23882.665} C_VEL
LIN {X 0,Y 165.599,Z 445.333,A -85,B 0,C 180,E1 -23884.583,E2 -23884.583} C_VEL
LIN {X 0,Y 168.355,Z 432.94,A -85,B 0,C 180,E1 -23886.315,E2 -23886.315} C_VEL
LIN {X 0,Y 170.407,Z 420.631,A -85,B 0,C 180,E1 -23887.559,E2 -23887.559} C_VEL
LIN {X 0,Y 171.787,Z 407.541,A -85,B 0,C 180,E1 -23888.469,E2 -23888.469} C_VEL
LIN {X 0,Y 173.005,Z 384.111,A -85,B 0,C 180,E1 -23889.419,E2 -23889.419} C_VEL
LIN {X 0,Y 171.162,Z 348.076,A -85,B 0,C 180,E1 -23891.682,E2 -23891.682} C_VEL
LIN {X 0,Y 169.938,Z 331.665,A -85,B 0,C 180,E1 -23892.853,E2 -23892.853} C_VEL
LIN {X 0,Y 164.694,Z 318.174,A -85,B 0,C 180,E1 -23895.06,E2 -23895.06} C_VEL
LIN {X 0,Y 158.451,Z 304.976,A -85,B 0,C 180,E1 -23897.814,E2 -23897.814} C_VEL
LIN {X 0,Y 154.196,Z 297.355,A -85,B 0,C 180,E1 -23899.812,E2 -23899.812} C_VEL
LIN {X 0,Y 152.227,Z 293.275,A -85,B 0,C 180,E1 -23901.022,E2 -23901.022} C_VEL
LIN {X 0,Y 150.207,Z 286.899,A -85,B 0,C 180,E1 -23905.387,E2 -23905.387} C_VEL
LIN {X 0,Y 150.182,Z 286.752,A -85,B 0,C 180,E1 -23909.019,E2 -23909.019} C_VEL
LIN {X 0,Y 150.233,Z 286.758,A -85,B 0,C 180,E1 -23912.722,E2 -23912.722} C_VEL
LIN {X 0,Y 150.278,Z 286.758,A -85,B 0,C 180,E1 -23919.275,E2 -23919.275} C_VEL
LIN {X 0,Y 150.311,Z 286.74,A -85,B 0,C 180,E1 -23923.708,E2 -23923.708} C_VEL
LIN {X 0,Y 150.599,Z 286.696,A -85,B 0,C 180,E1 -23929.242,E2 -23929.242} C_VEL
LIN {X 0,Y 150.673,Z 286.691,A -85,B 0,C 180,E1 -23931.957,E2 -23931.957} C_VEL
LIN {X 0,Y 151.187,Z 286.618,A -85,B 0,C 180,E1 -23940.001,E2 -23940.001} C_VEL
LIN {X 0,Y 150.67,Z 286.681,A -85,B 0,C 180,E1 -23948.045,E2 -23948.045} C_VEL
LIN {X 0,Y 150.567,Z 286.715,A -85,B 0,C 180,E1 -23951.428,E2 -23951.428} C_VEL
LIN {X 0,Y 150.313,Z 286.73,A -85,B 0,C 180,E1 -23956.293,E2 -23956.293} C_VEL
LIN {X 0,Y 150.277,Z 286.758,A -85,B 0,C 180,E1 -23960.723,E2 -23960.723} C_VEL
LIN {X 0,Y 150.177,Z 286.753,A -85,B 0,C 180,E1 -23967.237,E2 -23967.237} C_VEL
LIN {X 0,Y 150.197,Z 286.753,A -85,B 0,C 180,E1 -23972.625,E2 -23972.625} C_VEL
LIN {X 0,Y 150.165,Z 286.779,A -85,B 0,C 180,E1 -23977.477,E2 -23977.477} C_VEL
LIN {X 0,Y 150.127,Z 286.711,A -85,B 0,C 180,E1 -23981.498,E2 -23981.498} C_VEL
LIN {X 0,Y 150.13,Z 286.902,A -85,B 0,C 180,E1 -23987.023,E2 -23987.023} C_VEL
LIN {X 0,Y 150.383,Z 287.858,A -85,B 0,C 180,E1 -23987.759,E2 -23987.759} C_VEL
LIN {X 0,Y 151.926,Z 290.687,A -85,B 0,C 180,E1 -23988.636,E2 -23988.636} C_VEL
LIN {X 0,Y 153.576,Z 292.419,A -85,B 0,C 180,E1 -23989.396,E2 -23989.396} C_VEL
LIN {X 0,Y 155.845,Z 295.752,A -85,B 0,C 180,E1 -23990.461,E2 -23990.461} C_VEL
LIN {X 0,Y 161.61,Z 304.472,A -85,B 0,C 180,E1 -23992.97,E2 -23992.97} C_VEL
LIN {X 0,Y 168.817,Z 316.986,A -85,B 0,C 180,E1 -23995.835,E2 -23995.835} C_VEL
LIN {X 0,Y 175.708,Z 331.342,A -85,B 0,C 180,E1 -23998.382,E2 -23998.382} C_VEL
LIN {X 0,Y 173.78,Z 374.313,A -85,B 0,C 180,E1 -24000.16,E2 -24000.16} C_VEL
LIN {X 0,Y 172.797,Z 386.78,A -85,B 0,C 180,E1 -24001.122,E2 -24001.122} C_VEL
LIN {X 0,Y 171.164,Z 399.211,A -85,B 0,C 180,E1 -24002.49,E2 -24002.49} C_VEL
LIN {X 0,Y 169.027,Z 410.37,A -85,B 0,C 180,E1 -24004.116,E2 -24004.116} C_VEL
LIN {X 0,Y 166.354,Z 421.87,A -85,B 0,C 180,E1 -24006.339,E2 -24006.339} C_VEL
LIN {X 0,Y 163.607,Z 432.199,A -85,B 0,C 180,E1 -24008.916,E2 -24008.916} C_VEL
LIN {X 0,Y 161.031,Z 440.667,A -85,B 0,C 180,E1 -24011.555,E2 -24011.555} C_VEL
LIN {X 0,Y 158.456,Z 448.481,A -85,B 0,C 180,E1 -24014.568,E2 -24014.568} C_VEL
LIN {X 0,Y 155.77,Z 456.144,A -85,B 0,C 180,E1 -24018.287,E2 -24018.287} C_VEL
LIN {X 0,Y 153.647,Z 462.283,A -85,B 0,C 180,E1 -24022.114,E2 -24022.114} C_VEL
LIN {X 0,Y 152.008,Z 467.18,A -85,B 0,C 180,E1 -24026.024,E2 -24026.024} C_VEL
LIN {X 0,Y 150.783,Z 470.996,A -85,B 0,C 180,E1 -24030.001,E2 -24030.001} C_VEL
LIN {X 0,Y 150.314,Z 472.969,A -85,B 0,C 180,E1 -24032.681,E2 -24032.681} C_VEL
LIN {X 0,Y 150.247,Z 474.516,A -85,B 0,C 180,E1 -24035.369,E2 -24035.369} C_VEL
LIN {X 0,Y 150.269,Z 475.648,A -85,B 0,C 180,E1 -24038.067,E2 -24038.067} C_VEL
LIN {X 0,Y 150.972,Z 476.742,A -85,B 0,C 180,E1 -24043.46,E2 -24043.46} C_VEL
LIN {X 0,Y 151.673,Z 476.725,A -85,B 0,C 180,E1 -24046.143,E2 -24046.143} C_VEL
LIN {X 0,Y 152.661,Z 476.276,A -85,B 0,C 180,E1 -24048.8,E2 -24048.8} C_VEL
LIN {X 0,Y 155.419,Z 474.181,A -85,B 0,C 180,E1 -24054.016,E2 -24054.016} C_VEL
LIN {X 0,Y 158.106,Z 471.504,A -85,B 0,C 180,E1 -24057.823,E2 -24057.823} C_VEL
LIN {X 0,Y 161.367,Z 467.786,A -85,B 0,C 180,E1 -24061.509,E2 -24061.509} C_VEL
LIN {X 0,Y 165.17,Z 462.918,A -85,B 0,C 180,E1 -24065.06,E2 -24065.06} C_VEL
LIN {X 0,Y 169.477,Z 456.739,A -85,B 0,C 180,E1 -24068.465,E2 -24068.465} C_VEL
LIN {X 0,Y 174.297,Z 448.918,A -85,B 0,C 180,E1 -24071.706,E2 -24071.706} C_VEL
LIN {X 0,Y 178.609,Z 440.888,A -85,B 0,C 180,E1 -24074.302,E2 -24074.302} C_VEL
LIN {X 0,Y 183.107,Z 431.03,A -85,B 0,C 180,E1 -24076.824,E2 -24076.824} C_VEL
LIN {X 0,Y 187.402,Z 419.828,A -85,B 0,C 180,E1 -24079.002,E2 -24079.002} C_VEL
LIN {X 0,Y 190.871,Z 408.753,A -85,B 0,C 180,E1 -24080.645,E2 -24080.645} C_VEL
LIN {X 0,Y 193.476,Z 398.146,A -85,B 0,C 180,E1 -24081.864,E2 -24081.864} C_VEL
LIN {X 0,Y 195.537,Z 385.932,A -85,B 0,C 180,E1 -24082.965,E2 -24082.965} C_VEL
LIN {X 0,Y 196.824,Z 374.263,A -85,B 0,C 180,E1 -24083.674,E2 -24083.674} C_VEL
LIN {X 0,Y 198.025,Z 352.752,A -85,B 0,C 180,E1 -24084.516,E2 -24084.516} C_VEL
LIN {X 0,Y 192.817,Z 342.931,A -85,B 0,C 180,E1 -24087.07,E2 -24087.07} C_VEL
LIN {X 0,Y 187.458,Z 333.715,A -85,B 0,C 180,E1 -24089.974,E2 -24089.974} C_VEL
LIN {X 0,Y 182.465,Z 326.092,A -85,B 0,C 180,E1 -24093.003,E2 -24093.003} C_VEL
LIN {X 0,Y 179.75,Z 322.194,A -85,B 0,C 180,E1 -24094.83,E2 -24094.83} C_VEL
LIN {X 0,Y 177.147,Z 318.611,A -85,B 0,C 180,E1 -24096.732,E2 -24096.732} C_VEL
LIN {X 0,Y 173.985,Z 314.255,A -85,B 0,C 180,E1 -24099.315,E2 -24099.315} C_VEL
LIN {X 0,Y 171.302,Z 310.735,A -85,B 0,C 180,E1 -24101.798,E2 -24101.798} C_VEL
LIN {X 0,Y 170.653,Z 309.72,A -85,B 0,C 180,E1 -24102.473,E2 -24102.473} C_VEL
LIN {X 0,Y 168.035,Z 307.066,A -85,B 0,C 180,E1 -24105.311,E2 -24105.311} C_VEL
LIN {X 0,Y 166.651,Z 304.6,A -85,B 0,C 180,E1 -24107.208,E2 -24107.208} C_VEL
LIN {X 0,Y 163.992,Z 302.301,A -85,B 0,C 180,E1 -24111.295,E2 -24111.295} C_VEL
LIN {X 0,Y 162.46,Z 299.353,A -85,B 0,C 180,E1 -24115.036,E2 -24115.036} C_VEL
LIN {X 0,Y 161.187,Z 298.272,A -85,B 0,C 180,E1 -24119.999,E2 -24119.999} C_VEL
LIN {X 0,Y 162,Z 298.933,A -85,B 0,C 180,E1 -24129.993,E2 -24129.993} C_VEL
LIN {X 0,Y 162.531,Z 299.884,A -85,B 0,C 180,E1 -24131.69,E2 -24131.69} C_VEL
LIN {X 0,Y 164.052,Z 302.744,A -85,B 0,C 180,E1 -24135.291,E2 -24135.291} C_VEL
LIN {X 0,Y 165.494,Z 304.271,A -85,B 0,C 180,E1 -24137.677,E2 -24137.677} C_VEL
LIN {X 0,Y 168.109,Z 308.21,A -85,B 0,C 180,E1 -24141.296,E2 -24141.296} C_VEL
LIN {X 0,Y 172.917,Z 316.211,A -85,B 0,C 180,E1 -24146.451,E2 -24146.451} C_VEL
LIN {X 0,Y 177.039,Z 323.451,A -85,B 0,C 180,E1 -24149.996,E2 -24149.996} C_VEL
LIN {X 0,Y 180.341,Z 329.665,A -85,B 0,C 180,E1 -24152.483,E2 -24152.483} C_VEL
LIN {X 0,Y 184.044,Z 337.062,A -85,B 0,C 180,E1 -24154.999,E2 -24154.999} C_VEL
LIN {X 0,Y 189.136,Z 348.278,A -85,B 0,C 180,E1 -24158.122,E2 -24158.122} C_VEL
LIN {X 0,Y 193.564,Z 359.68,A -85,B 0,C 180,E1 -24160.629,E2 -24160.629} C_VEL
LIN {X 0,Y 194.899,Z 380.932,A -85,B 0,C 180,E1 -24162.363,E2 -24162.363} C_VEL
LIN {X 0,Y 195.259,Z 392.334,A -85,B 0,C 180,E1 -24163.134,E2 -24163.134} C_VEL
LIN {X 0,Y 193.727,Z 409.651,A -85,B 0,C 180,E1 -24163.77,E2 -24163.77} C_VEL
LIN {X 0,Y 191.651,Z 421.632,A -85,B 0,C 180,E1 -24164.452,E2 -24164.452} C_VEL
LIN {X 0,Y 188.912,Z 433.019,A -85,B 0,C 180,E1 -24165.397,E2 -24165.397} C_VEL
LIN {X 0,Y 184.944,Z 445.622,A -85,B 0,C 180,E1 -24166.842,E2 -24166.842} C_VEL
LIN {X 0,Y 180.439,Z 456.882,A -85,B 0,C 180,E1 -24168.536,E2 -24168.536} C_VEL
LIN {X 0,Y 175.661,Z 467.058,A -85,B 0,C 180,E1 -24170.569,E2 -24170.569} C_VEL
LIN {X 0,Y 170.205,Z 477.086,A -85,B 0,C 180,E1 -24173.221,E2 -24173.221} C_VEL
LIN {X 0,Y 164.95,Z 485.98,A -85,B 0,C 180,E1 -24176.365,E2 -24176.365} C_VEL
LIN {X 0,Y 160.286,Z 493.142,A -85,B 0,C 180,E1 -24179.719,E2 -24179.719} C_VEL
LIN {X 0,Y 156.362,Z 499.026,A -85,B 0,C 180,E1 -24183.363,E2 -24183.363} C_VEL
LIN {X 0,Y 153.252,Z 503.569,A -85,B 0,C 180,E1 -24187.057,E2 -24187.057} C_VEL
LIN {X 0,Y 150.965,Z 507.163,A -85,B 0,C 180,E1 -24190.981,E2 -24190.981} C_VEL
LIN {X 0,Y 149.702,Z 509.144,A -85,B 0,C 180,E1 -24193.931,E2 -24193.931} C_VEL
LIN {X 0,Y 148.456,Z 510.299,A -85,B 0,C 180,E1 -24196.119,E2 -24196.119} C_VEL
LIN {X 0,Y 145.138,Z 511.341,A -85,B 0,C 180,E1 -24199.749,E2 -24199.749} C_VEL
LIN {X 0,Y 142.77,Z 511.606,A -85,B 0,C 180,E1 -24202.776,E2 -24202.776} C_VEL
LIN {X 0,Y 142.002,Z 511.564,A -85,B 0,C 180,E1 -24205.145,E2 -24205.145} C_VEL
LIN {X 0,Y 142.051,Z 511.463,A -85,B 0,C 180,E1 -24205.943,E2 -24205.943} C_VEL
LIN {X 0,Y 142.672,Z 510.804,A -85,B 0,C 180,E1 -24209.999,E2 -24209.999} C_VEL
LIN {X 0,Y 142.278,Z 509.648,A -85,B 0,C 180,E1 -24212.83,E2 -24212.83} C_VEL
LIN {X 0,Y 141.738,Z 506.838,A -85,B 0,C 180,E1 -24217.393,E2 -24217.393} C_VEL
LIN {X 0,Y 141.934,Z 501.909,A -85,B 0,C 180,E1 -24222.873,E2 -24222.873} C_VEL
LIN {X 0,Y 143.175,Z 495.751,A -85,B 0,C 180,E1 -24227.864,E2 -24227.864} C_VEL
LIN {X 0,Y 145.147,Z 489.001,A -85,B 0,C 180,E1 -24232.038,E2 -24232.038} C_VEL
LIN {X 0,Y 148.005,Z 480.66,A -85,B 0,C 180,E1 -24236.053,E2 -24236.053} C_VEL
LIN {X 0,Y 150.911,Z 472.141,A -85,B 0,C 180,E1 -24239.272,E2 -24239.272} C_VEL
LIN {X 0,Y 154.041,Z 462.865,A -85,B 0,C 180,E1 -24242.029,E2 -24242.029} C_VEL
LIN {X 0,Y 156.798,Z 454.181,A -85,B 0,C 180,E1 -24244.073,E2 -24244.073} C_VEL
LIN {X 0,Y 159.807,Z 443.642,A -85,B 0,C 180,E1 -24246.027,E2 -24246.027} C_VEL
LIN {X 0,Y 162.448,Z 432.053,A -85,B 0,C 180,E1 -24247.666,E2 -24247.666} C_VEL
LIN {X 0,Y 164.667,Z 418.945,A -85,B 0,C 180,E1 -24249.013,E2 -24249.013} C_VEL
LIN {X 0,Y 166.033,Z 406.532,A -85,B 0,C 180,E1 -24249.873,E2 -24249.873} C_VEL
LIN {X 0,Y 167.224,Z 384.924,A -85,B 0,C 180,E1 -24250.769,E2 -24250.769} C_VEL
LIN {X 0,Y 165.518,Z 348.846,A -85,B 0,C 180,E1 -24253.134,E2 -24253.134} C_VEL
LIN {X 0,Y 164.474,Z 334.01,A -85,B 0,C 180,E1 -24254.242,E2 -24254.242} C_VEL
LIN {X 0,Y 159.779,Z 321.817,A -85,B 0,C 180,E1 -24256.368,E2 -24256.368} C_VEL
LIN {X 0,Y 154.146,Z 309.492,A -85,B 0,C 180,E1 -24259.05,E2 -24259.05} C_VEL
LIN {X 0,Y 149.599,Z 301.107,A -85,B 0,C 180,E1 -24261.359,E2 -24261.359} C_VEL
LIN {X 0,Y 147.263,Z 296.997,A -85,B 0,C 180,E1 -24262.628,E2 -24262.628} C_VEL
LIN {X 0,Y 144.598,Z 292.133,A -85,B 0,C 180,E1 -24264.322,E2 -24264.322} C_VEL
LIN {X 0,Y 143.188,Z 287.83,A -85,B 0,C 180,E1 -24267.532,E2 -24267.532} C_VEL
LIN {X 0,Y 143.177,Z 287.644,A -85,B 0,C 180,E1 -24272.069,E2 -24272.069} C_VEL
LIN {X 0,Y 143.219,Z 287.643,A -85,B 0,C 180,E1 -24278.799,E2 -24278.799} C_VEL
LIN {X 0,Y 143.25,Z 287.612,A -85,B 0,C 180,E1 -24282.881,E2 -24282.881} C_VEL
LIN {X 0,Y 143.526,Z 287.58,A -85,B 0,C 180,E1 -24288.705,E2 -24288.705} C_VEL
LIN {X 0,Y 143.599,Z 287.567,A -85,B 0,C 180,E1 -24291.558,E2 -24291.558} C_VEL
LIN {X 0,Y 144.146,Z 287.494,A -85,B 0,C 180,E1 -24300.001,E2 -24300.001} C_VEL
LIN {X 0,Y 143.597,Z 287.56,A -85,B 0,C 180,E1 -24308.444,E2 -24308.444} C_VEL
LIN {X 0,Y 143.493,Z 287.597,A -85,B 0,C 180,E1 -24311.616,E2 -24311.616} C_VEL
LIN {X 0,Y 143.251,Z 287.605,A -85,B 0,C 180,E1 -24317.12,E2 -24317.12} C_VEL
LIN {X 0,Y 143.214,Z 287.642,A -85,B 0,C 180,E1 -24321.195,E2 -24321.195} C_VEL
LIN {X 0,Y 143.133,Z 287.634,A -85,B 0,C 180,E1 -24327.898,E2 -24327.898} C_VEL
LIN {X 0,Y 143.129,Z 287.63,A -85,B 0,C 180,E1 -24333.415,E2 -24333.415} C_VEL
LIN {X 0,Y 143.047,Z 287.614,A -85,B 0,C 180,E1 -24339.696,E2 -24339.696} C_VEL
LIN {X 0,Y 143.103,Z 287.857,A -85,B 0,C 180,E1 -24344.055,E2 -24344.055} C_VEL
LIN {X 0,Y 143.39,Z 288.961,A -85,B 0,C 180,E1 -24344.744,E2 -24344.744} C_VEL
LIN {X 0,Y 145.068,Z 291.747,A -85,B 0,C 180,E1 -24345.781,E2 -24345.781} C_VEL
LIN {X 0,Y 146.62,Z 293.272,A -85,B 0,C 180,E1 -24346.594,E2 -24346.594} C_VEL
LIN {X 0,Y 148.709,Z 296.531,A -85,B 0,C 180,E1 -24347.725,E2 -24347.725} C_VEL
LIN {X 0,Y 150.072,Z 298.213,A -85,B 0,C 180,E1 -24348.404,E2 -24348.404} C_VEL
LIN {X 0,Y 155.583,Z 306.452,A -85,B 0,C 180,E1 -24351.046,E2 -24351.046} C_VEL
LIN {X 0,Y 161.2,Z 315.852,A -85,B 0,C 180,E1 -24353.509,E2 -24353.509} C_VEL
LIN {X 0,Y 166.484,Z 326.044,A -85,B 0,C 180,E1 -24355.673,E2 -24355.673} C_VEL
LIN {X 0,Y 169.988,Z 333.646,A -85,B 0,C 180,E1 -24357.043,E2 -24357.043} C_VEL
LIN {X 0,Y 167.971,Z 375.206,A -85,B 0,C 180,E1 -24358.802,E2 -24358.802} C_VEL
LIN {X 0,Y 166.924,Z 387.976,A -85,B 0,C 180,E1 -24359.829,E2 -24359.829} C_VEL
LIN {X 0,Y 165.183,Z 400.32,A -85,B 0,C 180,E1 -24361.231,E2 -24361.231} C_VEL
LIN {X 0,Y 162.781,Z 412.177,A -85,B 0,C 180,E1 -24363.044,E2 -24363.044} C_VEL
LIN {X 0,Y 159.991,Z 423.494,A -85,B 0,C 180,E1 -24365.337,E2 -24365.337} C_VEL
LIN {X 0,Y 157.098,Z 433.693,A -85,B 0,C 180,E1 -24367.998,E2 -24367.998} C_VEL
LIN {X 0,Y 154.382,Z 442.057,A -85,B 0,C 180,E1 -24370.73,E2 -24370.73} C_VEL
LIN {X 0,Y 151.129,Z 451.137,A -85,B 0,C 180,E1 -24374.492,E2 -24374.492} C_VEL
LIN {X 0,Y 148.407,Z 458.447,A -85,B 0,C 180,E1 -24378.391,E2 -24378.391} C_VEL
LIN {X 0,Y 146.024,Z 465.173,A -85,B 0,C 180,E1 -24383.091,E2 -24383.091} C_VEL
LIN {X 0,Y 144.493,Z 469.635,A -85,B 0,C 180,E1 -24387.213,E2 -24387.213} C_VEL
LIN {X 0,Y 143.701,Z 472.011,A -85,B 0,C 180,E1 -24390.001,E2 -24390.001} C_VEL
LIN {X 0,Y 143.251,Z 473.956,A -85,B 0,C 180,E1 -24392.813,E2 -24392.813} C_VEL
LIN {X 0,Y 143.208,Z 475.47,A -85,B 0,C 180,E1 -24395.634,E2 -24395.634} C_VEL
LIN {X 0,Y 143.52,Z 477.275,A -85,B 0,C 180,E1 -24401.297,E2 -24401.297} C_VEL
LIN {X 0,Y 144.856,Z 477.557,A -85,B 0,C 180,E1 -24406.925,E2 -24406.925} C_VEL
LIN {X 0,Y 147.245,Z 476.201,A -85,B 0,C 180,E1 -24412.448,E2 -24412.448} C_VEL
LIN {X 0,Y 150.618,Z 473.398,A -85,B 0,C 180,E1 -24417.554,E2 -24417.554} C_VEL
LIN {X 0,Y 154.085,Z 469.815,A -85,B 0,C 180,E1 -24421.637,E2 -24421.637} C_VEL
LIN {X 0,Y 157.948,Z 465.275,A -85,B 0,C 180,E1 -24425.342,E2 -24425.342} C_VEL
LIN {X 0,Y 162.717,Z 458.959,A -85,B 0,C 180,E1 -24429.137,E2 -24429.137} C_VEL
LIN {X 0,Y 167.268,Z 452.152,A -85,B 0,C 180,E1 -24432.242,E2 -24432.242} C_VEL
LIN {X 0,Y 171.742,Z 444.646,A -85,B 0,C 180,E1 -24434.903,E2 -24434.903} C_VEL
LIN {X 0,Y 175.775,Z 436.717,A -85,B 0,C 180,E1 -24437.178,E2 -24437.178} C_VEL
LIN {X 0,Y 180.26,Z 426.505,A -85,B 0,C 180,E1 -24439.488,E2 -24439.488} C_VEL
LIN {X 0,Y 184.274,Z 415.304,A -85,B 0,C 180,E1 -24441.43,E2 -24441.43} C_VEL
LIN {X 0,Y 187.854,Z 402.896,A -85,B 0,C 180,E1 -24443.043,E2 -24443.043} C_VEL
LIN {X 0,Y 190.206,Z 392.063,A -85,B 0,C 180,E1 -24444.088,E2 -24444.088} C_VEL
LIN {X 0,Y 191.809,Z 379.764,A -85,B 0,C 180,E1 -24445.027,E2 -24445.027} C_VEL
LIN {X 0,Y 193.012,Z 363.425,A -85,B 0,C 180,E1 -24445.751,E2 -24445.751} C_VEL
LIN {X 0,Y 193.403,Z 355.615,A -85,B 0,C 180,E1 -24446.068,E2 -24446.068} C_VEL
LIN {X 0,Y 187.799,Z 345.022,A -85,B 0,C 180,E1 -24449.059,E2 -24449.059} C_VEL
LIN {X 0,Y 182.788,Z 336.436,A -85,B 0,C 180,E1 -24452.056,E2 -24452.056} C_VEL
LIN {X 0,Y 177.863,Z 328.89,A -85,B 0,C 180,E1 -24455.396,E2 -24455.396} C_VEL
LIN {X 0,Y 174.854,Z 324.688,A -85,B 0,C 180,E1 -24457.698,E2 -24457.698} C_VEL
LIN {X 0,Y 172.039,Z 320.669,A -85,B 0,C 180,E1 -24460.134,E2 -24460.134} C_VEL
LIN {X 0,Y 168.883,Z 316.301,A -85,B 0,C 180,E1 -24463.289,E2 -24463.289} C_VEL
LIN {X 0,Y 166.39,Z 313.456,A -85,B 0,C 180,E1 -24466.197,E2 -24466.197} C_VEL
LIN {X 0,Y 165.347,Z 311.449,A -85,B 0,C 180,E1 -24467.729,E2 -24467.729} C_VEL
LIN {X 0,Y 162.841,Z 309.168,A -85,B 0,C 180,E1 -24471.78,E2 -24471.78} C_VEL
LIN {X 0,Y 161.481,Z 306.318,A -85,B 0,C 180,E1 -24475.319,E2 -24475.319} C_VEL
LIN {X 0,Y 160.317,Z 305.325,A -85,B 0,C 180,E1 -24479.999,E2 -24479.999} C_VEL
LIN {X 0,Y 161.14,Z 306.015,A -85,B 0,C 180,E1 -24490.047,E2 -24490.047} C_VEL
LIN {X 0,Y 163.094,Z 309.821,A -85,B 0,C 180,E1 -24495.183,E2 -24495.183} C_VEL
LIN {X 0,Y 164.208,Z 311.093,A -85,B 0,C 180,E1 -24497.112,E2 -24497.112} C_VEL
LIN {X 0,Y 166.418,Z 314.586,A -85,B 0,C 180,E1 -24500.379,E2 -24500.379} C_VEL
LIN {X 0,Y 170.974,Z 322.537,A -85,B 0,C 180,E1 -24505.597,E2 -24505.597} C_VEL
LIN {X 0,Y 174.702,Z 329.5,A -85,B 0,C 180,E1 -24509.019,E2 -24509.019} C_VEL
LIN {X 0,Y 177.839,Z 335.678,A -85,B 0,C 180,E1 -24511.533,E2 -24511.533} C_VEL
LIN {X 0,Y 181.958,Z 344.312,A -85,B 0,C 180,E1 -24514.48,E2 -24514.48} C_VEL
LIN {X 0,Y 186.703,Z 355.616,A -85,B 0,C 180,E1 -24517.542,E2 -24517.542} C_VEL
LIN {X 0,Y 189.37,Z 363.106,A -85,B 0,C 180,E1 -24519.173,E2 -24519.173} C_VEL
LIN {X 0,Y 190.625,Z 387.324,A -85,B 0,C 180,E1 -24521.161,E2 -24521.161} C_VEL
LIN {X 0,Y 190.712,Z 392.964,A -85,B 0,C 180,E1 -24521.53,E2 -24521.53} C_VEL
LIN {X 0,Y 189.151,Z 409.182,A -85,B 0,C 180,E1 -24522.129,E2 -24522.129} C_VEL
LIN {X 0,Y 186.874,Z 421.701,A -85,B 0,C 180,E1 -24522.868,E2 -24522.868} C_VEL
LIN {X 0,Y 183.941,Z 433.192,A -85,B 0,C 180,E1 -24523.849,E2 -24523.849} C_VEL
LIN {X 0,Y 179.841,Z 445.582,A -85,B 0,C 180,E1 -24525.298,E2 -24525.298} C_VEL
LIN {X 0,Y 175.184,Z 456.682,A -85,B 0,C 180,E1 -24527,E2 -24527} C_VEL
LIN {X 0,Y 169.706,Z 467.685,A -85,B 0,C 180,E1 -24529.288,E2 -24529.288} C_VEL
LIN {X 0,Y 164.576,Z 476.648,A -85,B 0,C 180,E1 -24531.742,E2 -24531.742} C_VEL
LIN {X 0,Y 159.064,Z 485.458,A -85,B 0,C 180,E1 -24534.943,E2 -24534.943} C_VEL
LIN {X 0,Y 154.159,Z 492.54,A -85,B 0,C 180,E1 -24538.38,E2 -24538.38} C_VEL
LIN {X 0,Y 150.07,Z 498.287,A -85,B 0,C 180,E1 -24542.074,E2 -24542.074} C_VEL
LIN {X 0,Y 147.113,Z 502.304,A -85,B 0,C 180,E1 -24545.403,E2 -24545.403} C_VEL
LIN {X 0,Y 144.22,Z 506.416,A -85,B 0,C 180,E1 -24550.054,E2 -24550.054} C_VEL
LIN {X 0,Y 142.101,Z 509.65,A -85,B 0,C 180,E1 -24555.682,E2 -24555.682} C_VEL
LIN {X 0,Y 141.672,Z 510.697,A -85,B 0,C 180,E1 -24558.554,E2 -24558.554} C_VEL
LIN {X 0,Y 141.708,Z 511.476,A -85,B 0,C 180,E1 -24562.699,E2 -24562.699} C_VEL
LIN {X 0,Y 142.051,Z 511.463,A -85,B 0,C 180,E1 -24565.943,E2 -24565.943} C_VEL
LIN {X 0,Y 141.93,Z 511.3,A -85,B 0,C 180,E1 -24567.519,E2 -24567.519} C_VEL
LIN {X 0,Y 140.65,Z 510.587,A -85,B 0,C 180,E1 -24569.844,E2 -24569.844} C_VEL
LIN {X 0,Y 137.235,Z 508.625,A -85,B 0,C 180,E1 -24573.669,E2 -24573.669} C_VEL
LIN {X 0,Y 135.001,Z 506.521,A -85,B 0,C 180,E1 -24576.86,E2 -24576.86} C_VEL
LIN {X 0,Y 134.606,Z 505.304,A -85,B 0,C 180,E1 -24578.507,E2 -24578.507} C_VEL
LIN {X 0,Y 134.93,Z 500.858,A -85,B 0,C 180,E1 -24583.554,E2 -24583.554} C_VEL
LIN {X 0,Y 136.365,Z 494.626,A -85,B 0,C 180,E1 -24588.789,E2 -24588.789} C_VEL
LIN {X 0,Y 138.53,Z 487.82,A -85,B 0,C 180,E1 -24593.15,E2 -24593.15} C_VEL
LIN {X 0,Y 141.592,Z 479.41,A -85,B 0,C 180,E1 -24597.329,E2 -24597.329} C_VEL
LIN {X 0,Y 144.697,Z 470.808,A -85,B 0,C 180,E1 -24600.661,E2 -24600.661} C_VEL
LIN {X 0,Y 148.518,Z 460.237,A -85,B 0,C 180,E1 -24603.779,E2 -24603.779} C_VEL
LIN {X 0,Y 152.225,Z 448.311,A -85,B 0,C 180,E1 -24606.469,E2 -24606.469} C_VEL
LIN {X 0,Y 154.965,Z 438.29,A -85,B 0,C 180,E1 -24608.162,E2 -24608.162} C_VEL
LIN {X 0,Y 157.593,Z 426.505,A -85,B 0,C 180,E1 -24609.661,E2 -24609.661} C_VEL
LIN {X 0,Y 159.631,Z 412.816,A -85,B 0,C 180,E1 -24610.909,E2 -24610.909} C_VEL
LIN {X 0,Y 160.857,Z 399.307,A -85,B 0,C 180,E1 -24611.657,E2 -24611.657} C_VEL
LIN {X 0,Y 161.517,Z 385.803,A -85,B 0,C 180,E1 -24612.218,E2 -24612.218} C_VEL
LIN {X 0,Y 160.093,Z 351.221,A -85,B 0,C 180,E1 -24614.564,E2 -24614.564} C_VEL
LIN {X 0,Y 159.271,Z 336.91,A -85,B 0,C 180,E1 -24615.644,E2 -24615.644} C_VEL
LIN {X 0,Y 155.124,Z 325.815,A -85,B 0,C 180,E1 -24617.677,E2 -24617.677} C_VEL
LIN {X 0,Y 149.848,Z 313.912,A -85,B 0,C 180,E1 -24620.391,E2 -24620.391} C_VEL
LIN {X 0,Y 144.296,Z 303.206,A -85,B 0,C 180,E1 -24623.496,E2 -24623.496} C_VEL
LIN {X 0,Y 140.08,Z 296.217,A -85,B 0,C 180,E1 -24626.075,E2 -24626.075} C_VEL
LIN {X 0,Y 136.653,Z 290.478,A -85,B 0,C 180,E1 -24628.62,E2 -24628.62} C_VEL
LIN {X 0,Y 136.082,Z 288.644,A -85,B 0,C 180,E1 -24630.294,E2 -24630.294} C_VEL
LIN {X 0,Y 136.117,Z 288.518,A -85,B 0,C 180,E1 -24632.311,E2 -24632.311} C_VEL
LIN {X 0,Y 136.183,Z 288.517,A -85,B 0,C 180,E1 -24638.824,E2 -24638.824} C_VEL
LIN {X 0,Y 136.222,Z 288.508,A -85,B 0,C 180,E1 -24645.051,E2 -24645.051} C_VEL
LIN {X 0,Y 136.419,Z 288.469,A -85,B 0,C 180,E1 -24648.178,E2 -24648.178} C_VEL
LIN {X 0,Y 136.528,Z 288.444,A -85,B 0,C 180,E1 -24651.117,E2 -24651.117} C_VEL
LIN {X 0,Y 137.103,Z 288.37,A -85,B 0,C 180,E1 -24660.001,E2 -24660.001} C_VEL
LIN {X 0,Y 136.527,Z 288.439,A -85,B 0,C 180,E1 -24668.885,E2 -24668.885} C_VEL
LIN {X 0,Y 136.408,Z 288.482,A -85,B 0,C 180,E1 -24671.894,E2 -24671.894} C_VEL
LIN {X 0,Y 136.162,Z 288.487,A -85,B 0,C 180,E1 -24678.041,E2 -24678.041} C_VEL
LIN {X 0,Y 136.138,Z 288.526,A -85,B 0,C 180,E1 -24681.691,E2 -24681.691} C_VEL
LIN {X 0,Y 136.053,Z 288.523,A -85,B 0,C 180,E1 -24688.584,E2 -24688.584} C_VEL
LIN {X 0,Y 136.035,Z 288.516,A -85,B 0,C 180,E1 -24694.633,E2 -24694.633} C_VEL
LIN {X 0,Y 136.005,Z 288.691,A -85,B 0,C 180,E1 -24700.145,E2 -24700.145} C_VEL
LIN {X 0,Y 136.224,Z 289.655,A -85,B 0,C 180,E1 -24700.984,E2 -24700.984} C_VEL
LIN {X 0,Y 137.6,Z 292.188,A -85,B 0,C 180,E1 -24702.051,E2 -24702.051} C_VEL
LIN {X 0,Y 139.815,Z 294.209,A -85,B 0,C 180,E1 -24703.408,E2 -24703.408} C_VEL
LIN {X 0,Y 142.072,Z 297.715,A -85,B 0,C 180,E1 -24704.82,E2 -24704.82} C_VEL
LIN {X 0,Y 143.283,Z 299.14,A -85,B 0,C 180,E1 -24705.508,E2 -24705.508} C_VEL
LIN {X 0,Y 145.932,Z 302.839,A -85,B 0,C 180,E1 -24706.985,E2 -24706.985} C_VEL
LIN {X 0,Y 151.403,Z 311.142,A -85,B 0,C 180,E1 -24709.8,E2 -24709.8} C_VEL
LIN {X 0,Y 157.034,Z 320.811,A -85,B 0,C 180,E1 -24712.444,E2 -24712.444} C_VEL
LIN {X 0,Y 162.093,Z 330.853,A -85,B 0,C 180,E1 -24714.655,E2 -24714.655} C_VEL
LIN {X 0,Y 164.383,Z 336.004,A -85,B 0,C 180,E1 -24715.622,E2 -24715.622} C_VEL
LIN {X 0,Y 162.369,Z 375.144,A -85,B 0,C 180,E1 -24717.296,E2 -24717.296} C_VEL
LIN {X 0,Y 161.331,Z 387.464,A -85,B 0,C 180,E1 -24718.276,E2 -24718.276} C_VEL
LIN {X 0,Y 159.478,Z 400.312,A -85,B 0,C 180,E1 -24719.735,E2 -24719.735} C_VEL
LIN {X 0,Y 156.954,Z 412.423,A -85,B 0,C 180,E1 -24721.593,E2 -24721.593} C_VEL
LIN {X 0,Y 154.013,Z 423.85,A -85,B 0,C 180,E1 -24723.948,E2 -24723.948} C_VEL
LIN {X 0,Y 150.95,Z 434.135,A -85,B 0,C 180,E1 -24726.689,E2 -24726.689} C_VEL
LIN {X 0,Y 147.768,Z 443.428,A -85,B 0,C 180,E1 -24729.831,E2 -24729.831} C_VEL
LIN {X 0,Y 144.353,Z 452.399,A -85,B 0,C 180,E1 -24733.745,E2 -24733.745} C_VEL
LIN {X 0,Y 141.523,Z 459.634,A -85,B 0,C 180,E1 -24737.817,E2 -24737.817} C_VEL
LIN {X 0,Y 139.025,Z 466.267,A -85,B 0,C 180,E1 -24742.741,E2 -24742.741} C_VEL
LIN {X 0,Y 137.446,Z 470.673,A -85,B 0,C 180,E1 -24747.07,E2 -24747.07} C_VEL
LIN {X 0,Y 136.621,Z 473.026,A -85,B 0,C 180,E1 -24750.001,E2 -24750.001} C_VEL
LIN {X 0,Y 136.189,Z 474.943,A -85,B 0,C 180,E1 -24752.959,E2 -24752.959} C_VEL
LIN {X 0,Y 136.152,Z 476.413,A -85,B 0,C 180,E1 -24755.927,E2 -24755.927} C_VEL
LIN {X 0,Y 136.568,Z 478.165,A -85,B 0,C 180,E1 -24761.88,E2 -24761.88} C_VEL
LIN {X 0,Y 137.151,Z 478.48,A -85,B 0,C 180,E1 -24764.846,E2 -24764.846} C_VEL
LIN {X 0,Y 138.044,Z 478.38,A -85,B 0,C 180,E1 -24767.787,E2 -24767.787} C_VEL
LIN {X 0,Y 140.668,Z 476.973,A -85,B 0,C 180,E1 -24773.56,E2 -24773.56} C_VEL
LIN {X 0,Y 144.191,Z 474.234,A -85,B 0,C 180,E1 -24778.675,E2 -24778.675} C_VEL
LIN {X 0,Y 148.043,Z 470.455,A -85,B 0,C 180,E1 -24783.089,E2 -24783.089} C_VEL
LIN {X 0,Y 152.158,Z 465.858,A -85,B 0,C 180,E1 -24786.903,E2 -24786.903} C_VEL
LIN {X 0,Y 157.082,Z 459.661,A -85,B 0,C 180,E1 -24790.691,E2 -24790.691} C_VEL
LIN {X 0,Y 162.05,Z 452.597,A -85,B 0,C 180,E1 -24793.941,E2 -24793.941} C_VEL
LIN {X 0,Y 166.743,Z 445.008,A -85,B 0,C 180,E1 -24796.641,E2 -24796.641} C_VEL
LIN {X 0,Y 171.693,Z 435.499,A -85,B 0,C 180,E1 -24799.313,E2 -24799.313} C_VEL
LIN {X 0,Y 176.222,Z 425.278,A -85,B 0,C 180,E1 -24801.506,E2 -24801.506} C_VEL
LIN {X 0,Y 180.437,Z 413.597,A -85,B 0,C 180,E1 -24803.45,E2 -24803.45} C_VEL
LIN {X 0,Y 183.64,Z 402.445,A -85,B 0,C 180,E1 -24804.828,E2 -24804.828} C_VEL
LIN {X 0,Y 186.153,Z 390.042,A -85,B 0,C 180,E1 -24806.008,E2 -24806.008} C_VEL
LIN {X 0,Y 187.678,Z 378.38,A -85,B 0,C 180,E1 -24806.81,E2 -24806.81} C_VEL
LIN {X 0,Y 189.055,Z 358.851,A -85,B 0,C 180,E1 -24807.617,E2 -24807.617} C_VEL
LIN {X 0,Y 183.199,Z 347.643,A -85,B 0,C 180,E1 -24811.031,E2 -24811.031} C_VEL
LIN {X 0,Y 178.092,Z 338.912,A -85,B 0,C 180,E1 -24814.429,E2 -24814.429} C_VEL
LIN {X 0,Y 173.296,Z 331.596,A -85,B 0,C 180,E1 -24818.123,E2 -24818.123} C_VEL
LIN {X 0,Y 170.089,Z 327.022,A -85,B 0,C 180,E1 -24821.01,E2 -24821.01} C_VEL
LIN {X 0,Y 167.142,Z 322.829,A -85,B 0,C 180,E1 -24824.138,E2 -24824.138} C_VEL
LIN {X 0,Y 164.709,Z 319.738,A -85,B 0,C 180,E1 -24827.211,E2 -24827.211} C_VEL
LIN {X 0,Y 163.841,Z 318.21,A -85,B 0,C 180,E1 -24828.557,E2 -24828.557} C_VEL
LIN {X 0,Y 161.192,Z 315.176,A -85,B 0,C 180,E1 -24833.467,E2 -24833.467} C_VEL
LIN {X 0,Y 160.431,Z 313.244,A -85,B 0,C 180,E1 -24835.82,E2 -24835.82} C_VEL
LIN {X 0,Y 159.447,Z 312.377,A -85,B 0,C 180,E1 -24839.999,E2 -24839.999} C_VEL
LIN {X 0,Y 160.092,Z 312.978,A -85,B 0,C 180,E1 -24849.475,E2 -24849.475} C_VEL
LIN {X 0,Y 160.41,Z 313.702,A -85,B 0,C 180,E1 -24850.674,E2 -24850.674} C_VEL
LIN {X 0,Y 161.902,Z 316.63,A -85,B 0,C 180,E1 -24854.614,E2 -24854.614} C_VEL
LIN {X 0,Y 162.979,Z 317.972,A -85,B 0,C 180,E1 -24856.599,E2 -24856.599} C_VEL
LIN {X 0,Y 164.876,Z 321.169,A -85,B 0,C 180,E1 -24859.593,E2 -24859.593} C_VEL
LIN {X 0,Y 169.035,Z 328.877,A -85,B 0,C 180,E1 -24864.696,E2 -24864.696} C_VEL
LIN {X 0,Y 172.374,Z 335.417,A -85,B 0,C 180,E1 -24867.972,E2 -24867.972} C_VEL
LIN {X 0,Y 175.171,Z 341.222,A -85,B 0,C 180,E1 -24870.38,E2 -24870.38} C_VEL
LIN {X 0,Y 178.93,Z 349.536,A -85,B 0,C 180,E1 -24873.275,E2 -24873.275} C_VEL
LIN {X 0,Y 183.263,Z 360.332,A -85,B 0,C 180,E1 -24876.284,E2 -24876.284} C_VEL
LIN {X 0,Y 185.297,Z 366.093,A -85,B 0,C 180,E1 -24877.619,E2 -24877.619} C_VEL
LIN {X 0,Y 186.311,Z 390.107,A -85,B 0,C 180,E1 -24879.623,E2 -24879.623} C_VEL
LIN {X 0,Y 186.219,Z 394.889,A -85,B 0,C 180,E1 -24879.888,E2 -24879.888} C_VEL
LIN {X 0,Y 184.687,Z 409.224,A -85,B 0,C 180,E1 -24880.441,E2 -24880.441} C_VEL
LIN {X 0,Y 182.254,Z 421.728,A -85,B 0,C 180,E1 -24881.201,E2 -24881.201} C_VEL
LIN {X 0,Y 179.116,Z 433.38,A -85,B 0,C 180,E1 -24882.217,E2 -24882.217} C_VEL
LIN {X 0,Y 174.874,Z 445.557,A -85,B 0,C 180,E1 -24883.664,E2 -24883.664} C_VEL
LIN {X 0,Y 170.065,Z 456.454,A -85,B 0,C 180,E1 -24885.369,E2 -24885.369} C_VEL
LIN {X 0,Y 164.395,Z 467.338,A -85,B 0,C 180,E1 -24887.676,E2 -24887.676} C_VEL
LIN {X 0,Y 159.069,Z 476.215,A -85,B 0,C 180,E1 -24890.16,E2 -24890.16} C_VEL
LIN {X 0,Y 153.279,Z 484.922,A -85,B 0,C 180,E1 -24893.411,E2 -24893.411} C_VEL
LIN {X 0,Y 148.137,Z 491.941,A -85,B 0,C 180,E1 -24896.935,E2 -24896.935} C_VEL
LIN {X 0,Y 143.791,Z 497.633,A -85,B 0,C 180,E1 -24900.74,E2 -24900.74} C_VEL
LIN {X 0,Y 140.336,Z 501.968,A -85,B 0,C 180,E1 -24904.57,E2 -24904.57} C_VEL
LIN {X 0,Y 137.519,Z 505.669,A -85,B 0,C 180,E1 -24909.038,E2 -24909.038} C_VEL
LIN {X 0,Y 135.184,Z 508.861,A -85,B 0,C 180,E1 -24914.932,E2 -24914.932} C_VEL
LIN {X 0,Y 134.659,Z 509.875,A -85,B 0,C 180,E1 -24917.949,E2 -24917.949} C_VEL
LIN {X 0,Y 134.645,Z 510.661,A -85,B 0,C 180,E1 -24922.624,E2 -24922.624} C_VEL
LIN {X 0,Y 135.2,Z 510.509,A -85,B 0,C 180,E1 -24927.019,E2 -24927.019} C_VEL
LIN {X 0,Y 135.617,Z 509.902,A -85,B 0,C 180,E1 -24929.999,E2 -24929.999} C_VEL
LIN {X 0,Y 135.187,Z 508.7,A -85,B 0,C 180,E1 -24932.979,E2 -24932.979} C_VEL
LIN {X 0,Y 134.606,Z 505.304,A -85,B 0,C 180,E1 -24938.507,E2 -24938.507} C_VEL
LIN {X 0,Y 133.975,Z 503.366,A -85,B 0,C 180,E1 -24940.873,E2 -24940.873} C_VEL
LIN {X 0,Y 131.601,Z 499.579,A -85,B 0,C 180,E1 -24944.695,E2 -24944.695} C_VEL
LIN {X 0,Y 129.744,Z 495.157,A -85,B 0,C 180,E1 -24948.515,E2 -24948.515} C_VEL
LIN {X 0,Y 129.941,Z 492.192,A -85,B 0,C 180,E1 -24950.782,E2 -24950.782} C_VEL
LIN {X 0,Y 132.822,Z 484.357,A -85,B 0,C 180,E1 -24955.668,E2 -24955.668} C_VEL
LIN {X 0,Y 136.593,Z 474.876,A -85,B 0,C 180,E1 -24960.107,E2 -24960.107} C_VEL
LIN {X 0,Y 140.134,Z 465.475,A -85,B 0,C 180,E1 -24963.479,E2 -24963.479} C_VEL
LIN {X 0,Y 143.861,Z 455.043,A -85,B 0,C 180,E1 -24966.321,E2 -24966.321} C_VEL
LIN {X 0,Y 147.556,Z 443.5,A -85,B 0,C 180,E1 -24968.69,E2 -24968.69} C_VEL
LIN {X 0,Y 150.674,Z 431.405,A -85,B 0,C 180,E1 -24970.546,E2 -24970.546} C_VEL
LIN {X 0,Y 153.056,Z 418.833,A -85,B 0,C 180,E1 -24971.937,E2 -24971.937} C_VEL
LIN {X 0,Y 154.724,Z 405.405,A -85,B 0,C 180,E1 -24972.946,E2 -24972.946} C_VEL
LIN {X 0,Y 155.925,Z 386.626,A -85,B 0,C 180,E1 -24973.774,E2 -24973.774} C_VEL
LIN {X 0,Y 154.712,Z 352.417,A -85,B 0,C 180,E1 -24976.185,E2 -24976.185} C_VEL
LIN {X 0,Y 154.061,Z 339.539,A -85,B 0,C 180,E1 -24977.193,E2 -24977.193} C_VEL
LIN {X 0,Y 150.412,Z 329.42,A -85,B 0,C 180,E1 -24979.145,E2 -24979.145} C_VEL
LIN {X 0,Y 145.49,Z 318.074,A -85,B 0,C 180,E1 -24981.89,E2 -24981.89} C_VEL
LIN {X 0,Y 140.42,Z 307.976,A -85,B 0,C 180,E1 -24984.97,E2 -24984.97} C_VEL
LIN {X 0,Y 136.705,Z 301.502,A -85,B 0,C 180,E1 -24987.44,E2 -24987.44} C_VEL
LIN {X 0,Y 132.888,Z 295.403,A -85,B 0,C 180,E1 -24990.239,E2 -24990.239} C_VEL
LIN {X 0,Y 129.939,Z 292.049,A -85,B 0,C 180,E1 -24992.521,E2 -24992.521} C_VEL
LIN {X 0,Y 129.14,Z 290.081,A -85,B 0,C 180,E1 -24993.54,E2 -24993.54} C_VEL
LIN {X 0,Y 129.001,Z 289.442,A -85,B 0,C 180,E1 -24994.594,E2 -24994.594} C_VEL
LIN {X 0,Y 129.065,Z 289.404,A -85,B 0,C 180,E1 -24997.769,E2 -24997.769} C_VEL
LIN {X 0,Y 129.143,Z 289.377,A -85,B 0,C 180,E1 -25004.211,E2 -25004.211} C_VEL
LIN {X 0,Y 129.338,Z 289.351,A -85,B 0,C 180,E1 -25007.972,E2 -25007.972} C_VEL
LIN {X 0,Y 129.454,Z 289.323,A -85,B 0,C 180,E1 -25010.627,E2 -25010.627} C_VEL
LIN {X 0,Y 130.058,Z 289.246,A -85,B 0,C 180,E1 -25020.001,E2 -25020.001} C_VEL
LIN {X 0,Y 129.453,Z 289.32,A -85,B 0,C 180,E1 -25029.374,E2 -25029.374} C_VEL
LIN {X 0,Y 129.292,Z 289.375,A -85,B 0,C 180,E1 -25032.559,E2 -25032.559} C_VEL
LIN {X 0,Y 129.076,Z 289.373,A -85,B 0,C 180,E1 -25039.069,E2 -25039.069} C_VEL
LIN {X 0,Y 129.029,Z 289.409,A -85,B 0,C 180,E1 -25042.414,E2 -25042.414} C_VEL
LIN {X 0,Y 128.976,Z 289.414,A -85,B 0,C 180,E1 -25049.369,E2 -25049.369} C_VEL
LIN {X 0,Y 128.952,Z 289.493,A -85,B 0,C 180,E1 -25055.386,E2 -25055.386} C_VEL
LIN {X 0,Y 129.114,Z 290.373,A -85,B 0,C 180,E1 -25056.418,E2 -25056.418} C_VEL
LIN {X 0,Y 130.515,Z 293.044,A -85,B 0,C 180,E1 -25057.773,E2 -25057.773} C_VEL
LIN {X 0,Y 132.972,Z 295.182,A -85,B 0,C 180,E1 -25059.591,E2 -25059.591} C_VEL
LIN {X 0,Y 135.096,Z 298.523,A -85,B 0,C 180,E1 -25061.18,E2 -25061.18} C_VEL
LIN {X 0,Y 136.847,Z 300.414,A -85,B 0,C 180,E1 -25062.337,E2 -25062.337} C_VEL
LIN {X 0,Y 139.607,Z 304.194,A -85,B 0,C 180,E1 -25064.109,E2 -25064.109} C_VEL
LIN {X 0,Y 145.925,Z 313.649,A -85,B 0,C 180,E1 -25067.759,E2 -25067.759} C_VEL
LIN {X 0,Y 150.993,Z 322.221,A -85,B 0,C 180,E1 -25070.377,E2 -25070.377} C_VEL
LIN {X 0,Y 156.637,Z 333.174,A -85,B 0,C 180,E1 -25073.065,E2 -25073.065} C_VEL
LIN {X 0,Y 158.813,Z 338.11,A -85,B 0,C 180,E1 -25074.064,E2 -25074.064} C_VEL
LIN {X 0,Y 156.721,Z 376.888,A -85,B 0,C 180,E1 -25075.802,E2 -25075.802} C_VEL
LIN {X 0,Y 155.494,Z 389.904,A -85,B 0,C 180,E1 -25076.908,E2 -25076.908} C_VEL
LIN {X 0,Y 153.496,Z 402.487,A -85,B 0,C 180,E1 -25078.423,E2 -25078.423} C_VEL
LIN {X 0,Y 150.839,Z 414.215,A -85,B 0,C 180,E1 -25080.329,E2 -25080.329} C_VEL
LIN {X 0,Y 147.763,Z 425.466,A -85,B 0,C 180,E1 -25082.757,E2 -25082.757} C_VEL
LIN {X 0,Y 144.559,Z 435.615,A -85,B 0,C 180,E1 -25085.593,E2 -25085.593} C_VEL
LIN {X 0,Y 141.194,Z 444.765,A -85,B 0,C 180,E1 -25088.848,E2 -25088.848} C_VEL
LIN {X 0,Y 137.638,Z 453.648,A -85,B 0,C 180,E1 -25092.928,E2 -25092.928} C_VEL
LIN {X 0,Y 134.64,Z 460.819,A -85,B 0,C 180,E1 -25097.184,E2 -25097.184} C_VEL
LIN {X 0,Y 132.768,Z 465.646,A -85,B 0,C 180,E1 -25100.864,E2 -25100.864} C_VEL
LIN {X 0,Y 130.88,Z 470.38,A -85,B 0,C 180,E1 -25105.381,E2 -25105.381} C_VEL
LIN {X 0,Y 129.542,Z 474.038,A -85,B 0,C 180,E1 -25110.001,E2 -25110.001} C_VEL
LIN {X 0,Y 129.126,Z 475.928,A -85,B 0,C 180,E1 -25113.121,E2 -25113.121} C_VEL
LIN {X 0,Y 129.088,Z 477.353,A -85,B 0,C 180,E1 -25116.252,E2 -25116.252} C_VEL
LIN {X 0,Y 129.627,Z 479.069,A -85,B 0,C 180,E1 -25122.599,E2 -25122.599} C_VEL
LIN {X 0,Y 130.282,Z 479.345,A -85,B 0,C 180,E1 -25125.649,E2 -25125.649} C_VEL
LIN {X 0,Y 131.277,Z 479.2,A -85,B 0,C 180,E1 -25128.737,E2 -25128.737} C_VEL
LIN {X 0,Y 134.149,Z 477.746,A -85,B 0,C 180,E1 -25134.779,E2 -25134.779} C_VEL
LIN {X 0,Y 137.698,Z 475.145,A -85,B 0,C 180,E1 -25139.81,E2 -25139.81} C_VEL
LIN {X 0,Y 142.1,Z 471.098,A -85,B 0,C 180,E1 -25144.665,E2 -25144.665} C_VEL
LIN {X 0,Y 146.498,Z 466.441,A -85,B 0,C 180,E1 -25148.584,E2 -25148.584} C_VEL
LIN {X 0,Y 151.589,Z 460.353,A -85,B 0,C 180,E1 -25152.359,E2 -25152.359} C_VEL
LIN {X 0,Y 156.976,Z 453.043,A -85,B 0,C 180,E1 -25155.753,E2 -25155.753} C_VEL
LIN {X 0,Y 161.907,Z 445.363,A -85,B 0,C 180,E1 -25158.485,E2 -25158.485} C_VEL
LIN {X 0,Y 167.01,Z 435.918,A -85,B 0,C 180,E1 -25161.122,E2 -25161.122} C_VEL
LIN {X 0,Y 171.839,Z 425.344,A -85,B 0,C 180,E1 -25163.382,E2 -25163.382} C_VEL
LIN {X 0,Y 175.69,Z 415.077,A -85,B 0,C 180,E1 -25165.089,E2 -25165.089} C_VEL
LIN {X 0,Y 179.237,Z 403.337,A -85,B 0,C 180,E1 -25166.557,E2 -25166.557} C_VEL
LIN {X 0,Y 181.878,Z 390.908,A -85,B 0,C 180,E1 -25167.742,E2 -25167.742} C_VEL
LIN {X 0,Y 183.517,Z 378.755,A -85,B 0,C 180,E1 -25168.584,E2 -25168.584} C_VEL
LIN {X 0,Y 184.695,Z 361.874,A -85,B 0,C 180,E1 -25169.325,E2 -25169.325} C_VEL
LIN {X 0,Y 179.808,Z 352.272,A -85,B 0,C 180,E1 -25172.423,E2 -25172.423} C_VEL
LIN {X 0,Y 175.512,Z 344.707,A -85,B 0,C 180,E1 -25175.486,E2 -25175.486} C_VEL
LIN {X 0,Y 171.151,Z 337.78,A -85,B 0,C 180,E1 -25179.063,E2 -25179.063} C_VEL
LIN {X 0,Y 168.107,Z 333.27,A -85,B 0,C 180,E1 -25181.982,E2 -25181.982} C_VEL
LIN {X 0,Y 165.537,Z 329.41,A -85,B 0,C 180,E1 -25184.894,E2 -25184.894} C_VEL
LIN {X 0,Y 163.198,Z 326.24,A -85,B 0,C 180,E1 -25188.058,E2 -25188.058} C_VEL
LIN {X 0,Y 162.572,Z 325.065,A -85,B 0,C 180,E1 -25189.097,E2 -25189.097} C_VEL
LIN {X 0,Y 159.971,Z 321.779,A -85,B 0,C 180,E1 -25194.327,E2 -25194.327} C_VEL
LIN {X 0,Y 159.302,Z 320.068,A -85,B 0,C 180,E1 -25196.642,E2 -25196.642} C_VEL
LIN {X 0,Y 158.577,Z 319.428,A -85,B 0,C 180,E1 -25199.999,E2 -25199.999} C_VEL
LIN {X 0,Y 159.23,Z 320.069,A -85,B 0,C 180,E1 -25209.527,E2 -25209.527} C_VEL
LIN {X 0,Y 160.634,Z 323.34,A -85,B 0,C 180,E1 -25213.843,E2 -25213.843} C_VEL
LIN {X 0,Y 161.783,Z 324.888,A -85,B 0,C 180,E1 -25216.117,E2 -25216.117} C_VEL
LIN {X 0,Y 163.449,Z 327.919,A -85,B 0,C 180,E1 -25218.923,E2 -25218.923} C_VEL
LIN {X 0,Y 167.035,Z 334.975,A -85,B 0,C 180,E1 -25223.647,E2 -25223.647} C_VEL
LIN {X 0,Y 170.08,Z 341.29,A -85,B 0,C 180,E1 -25226.873,E2 -25226.873} C_VEL
LIN {X 0,Y 172.781,Z 347.238,A -85,B 0,C 180,E1 -25229.373,E2 -25229.373} C_VEL
LIN {X 0,Y 176.023,Z 354.794,A -85,B 0,C 180,E1 -25232.055,E2 -25232.055} C_VEL
LIN {X 0,Y 180.158,Z 365.729,A -85,B 0,C 180,E1 -25235.154,E2 -25235.154} C_VEL
LIN {X 0,Y 181.332,Z 369.169,A -85,B 0,C 180,E1 -25235.985,E2 -25235.985} C_VEL
LIN {X 0,Y 182.094,Z 392.548,A -85,B 0,C 180,E1 -25237.971,E2 -25237.971} C_VEL
LIN {X 0,Y 180.852,Z 406.07,A -85,B 0,C 180,E1 -25238.528,E2 -25238.528} C_VEL
LIN {X 0,Y 178.338,Z 419.551,A -85,B 0,C 180,E1 -25239.284,E2 -25239.284} C_VEL
LIN {X 0,Y 175.076,Z 431.581,A -85,B 0,C 180,E1 -25240.297,E2 -25240.297} C_VEL
LIN {X 0,Y 170.672,Z 443.947,A -85,B 0,C 180,E1 -25241.724,E2 -25241.724} C_VEL
LIN {X 0,Y 165.715,Z 455.026,A -85,B 0,C 180,E1 -25243.425,E2 -25243.425} C_VEL
LIN {X 0,Y 160.349,Z 465.026,A -85,B 0,C 180,E1 -25245.471,E2 -25245.471} C_VEL
LIN {X 0,Y 154.73,Z 474.137,A -85,B 0,C 180,E1 -25247.936,E2 -25247.936} C_VEL
LIN {X 0,Y 148.597,Z 483.082,A -85,B 0,C 180,E1 -25251.195,E2 -25251.195} C_VEL
LIN {X 0,Y 143.084,Z 490.312,A -85,B 0,C 180,E1 -25254.75,E2 -25254.75} C_VEL
LIN {X 0,Y 137.619,Z 496.985,A -85,B 0,C 180,E1 -25259.29,E2 -25259.29} C_VEL
LIN {X 0,Y 134.363,Z 500.821,A -85,B 0,C 180,E1 -25262.773,E2 -25262.773} C_VEL
LIN {X 0,Y 130.836,Z 504.92,A -85,B 0,C 180,E1 -25267.912,E2 -25267.912} C_VEL
LIN {X 0,Y 128.302,Z 508.073,A -85,B 0,C 180,E1 -25274.103,E2 -25274.103} C_VEL
LIN {X 0,Y 127.515,Z 509.624,A -85,B 0,C 180,E1 -25280.482,E2 -25280.482} C_VEL
LIN {X 0,Y 128.104,Z 509.622,A -85,B 0,C 180,E1 -25286.854,E2 -25286.854} C_VEL
LIN {X 0,Y 128.559,Z 508.99,A -85,B 0,C 180,E1 -25289.999,E2 -25289.999} C_VEL
LIN {X 0,Y 128.077,Z 507.749,A -85,B 0,C 180,E1 -25293.144,E2 -25293.144} C_VEL
LIN {X 0,Y 127.547,Z 504.717,A -85,B 0,C 180,E1 -25298.394,E2 -25298.394} C_VEL
LIN {X 0,Y 127.963,Z 499.81,A -85,B 0,C 180,E1 -25304.307,E2 -25304.307} C_VEL
LIN {X 0,Y 129.542,Z 493.493,A -85,B 0,C 180,E1 -25309.819,E2 -25309.819} C_VEL
LIN {X 0,Y 129.941,Z 492.192,A -85,B 0,C 180,E1 -25310.782,E2 -25310.782} C_VEL
LIN {X 0,Y 130.359,Z 489.06,A -85,B 0,C 180,E1 -25312.986,E2 -25312.986} C_VEL
LIN {X 0,Y 129.773,Z 483.467,A -85,B 0,C 180,E1 -25316.589,E2 -25316.589} C_VEL
LIN {X 0,Y 129.577,Z 477.271,A -85,B 0,C 180,E1 -25320.011,E2 -25320.011} C_VEL
LIN {X 0,Y 130.569,Z 473.197,A -85,B 0,C 180,E1 -25321.848,E2 -25321.848} C_VEL
LIN {X 0,Y 134.595,Z 462.957,A -85,B 0,C 180,E1 -25325.511,E2 -25325.511} C_VEL
LIN {X 0,Y 137.711,Z 454.806,A -85,B 0,C 180,E1 -25327.762,E2 -25327.762} C_VEL
LIN {X 0,Y 141.573,Z 443.406,A -85,B 0,C 180,E1 -25330.189,E2 -25330.189} C_VEL
LIN {X 0,Y 144.817,Z 431.547,A -85,B 0,C 180,E1 -25332.089,E2 -25332.089} C_VEL
LIN {X 0,Y 147.36,Z 419.016,A -85,B 0,C 180,E1 -25333.55,E2 -25333.55} C_VEL
LIN {X 0,Y 149.144,Z 405.75,A -85,B 0,C 180,E1 -25334.599,E2 -25334.599} C_VEL
LIN {X 0,Y 150.461,Z 387.511,A -85,B 0,C 180,E1 -25335.437,E2 -25335.437} C_VEL
LIN {X 0,Y 149.464,Z 353.863,A -85,B 0,C 180,E1 -25337.905,E2 -25337.905} C_VEL
LIN {X 0,Y 148.916,Z 341.739,A -85,B 0,C 180,E1 -25338.898,E2 -25338.898} C_VEL
LIN {X 0,Y 145.06,Z 331.026,A -85,B 0,C 180,E1 -25341.155,E2 -25341.155} C_VEL
LIN {X 0,Y 140.111,Z 319.756,A -85,B 0,C 180,E1 -25344.203,E2 -25344.203} C_VEL
LIN {X 0,Y 136.039,Z 311.675,A -85,B 0,C 180,E1 -25346.943,E2 -25346.943} C_VEL
LIN {X 0,Y 133.054,Z 306.315,A -85,B 0,C 180,E1 -25349.127,E2 -25349.127} C_VEL
LIN {X 0,Y 129.915,Z 300.973,A -85,B 0,C 180,E1 -25351.639,E2 -25351.639} C_VEL
LIN {X 0,Y 127.321,Z 297.996,A -85,B 0,C 180,E1 -25353.795,E2 -25353.795} C_VEL
LIN {X 0,Y 126.211,Z 295.954,A -85,B 0,C 180,E1 -25354.876,E2 -25354.876} C_VEL
LIN {X 0,Y 123.691,Z 294.066,A -85,B 0,C 180,E1 -25357.208,E2 -25357.208} C_VEL
LIN {X 0,Y 122.167,Z 291.236,A -85,B 0,C 180,E1 -25359.109,E2 -25359.109} C_VEL
LIN {X 0,Y 122.032,Z 290.385,A -85,B 0,C 180,E1 -25360.443,E2 -25360.443} C_VEL
LIN {X 0,Y 122.281,Z 290.232,A -85,B 0,C 180,E1 -25367.693,E2 -25367.693} C_VEL
LIN {X 0,Y 122.383,Z 290.203,A -85,B 0,C 180,E1 -25370.08,E2 -25370.08} C_VEL
LIN {X 0,Y 122.55,Z 290.194,A -85,B 0,C 180,E1 -25376.713,E2 -25376.713} C_VEL
LIN {X 0,Y 123.011,Z 290.123,A -85,B 0,C 180,E1 -25380.001,E2 -25380.001} C_VEL
LIN {X 0,Y 122.371,Z 290.206,A -85,B 0,C 180,E1 -25386.969,E2 -25386.969} C_VEL
LIN {X 0,Y 122.281,Z 290.243,A -85,B 0,C 180,E1 -25392.309,E2 -25392.309} C_VEL
LIN {X 0,Y 122.056,Z 290.242,A -85,B 0,C 180,E1 -25396.733,E2 -25396.733} C_VEL
LIN {X 0,Y 121.974,Z 290.28,A -85,B 0,C 180,E1 -25402.801,E2 -25402.801} C_VEL
LIN {X 0,Y 121.946,Z 290.525,A -85,B 0,C 180,E1 -25409.697,E2 -25409.697} C_VEL
LIN {X 0,Y 122.163,Z 291.62,A -85,B 0,C 180,E1 -25410.802,E2 -25410.802} C_VEL
LIN {X 0,Y 123.559,Z 294.041,A -85,B 0,C 180,E1 -25412.467,E2 -25412.467} C_VEL
LIN {X 0,Y 126.346,Z 296.334,A -85,B 0,C 180,E1 -25415.069,E2 -25415.069} C_VEL
LIN {X 0,Y 128.272,Z 299.472,A -85,B 0,C 180,E1 -25416.855,E2 -25416.855} C_VEL
LIN {X 0,Y 130.253,Z 301.408,A -85,B 0,C 180,E1 -25418.428,E2 -25418.428} C_VEL
LIN {X 0,Y 132.681,Z 304.898,A -85,B 0,C 180,E1 -25420.314,E2 -25420.314} C_VEL
LIN {X 0,Y 134.193,Z 306.835,A -85,B 0,C 180,E1 -25421.393,E2 -25421.393} C_VEL
LIN {X 0,Y 137.501,Z 311.681,A -85,B 0,C 180,E1 -25423.633,E2 -25423.633} C_VEL
LIN {X 0,Y 142.091,Z 318.621,A -85,B 0,C 180,E1 -25426.428,E2 -25426.428} C_VEL
LIN {X 0,Y 146.701,Z 326.619,A -85,B 0,C 180,E1 -25428.996,E2 -25428.996} C_VEL
LIN {X 0,Y 152.101,Z 337.396,A -85,B 0,C 180,E1 -25431.769,E2 -25431.769} C_VEL
LIN {X 0,Y 153.326,Z 340.313,A -85,B 0,C 180,E1 -25432.385,E2 -25432.385} C_VEL
LIN {X 0,Y 151.295,Z 377.395,A -85,B 0,C 180,E1 -25434.112,E2 -25434.112} C_VEL
LIN {X 0,Y 150.022,Z 390.223,A -85,B 0,C 180,E1 -25435.214,E2 -25435.214} C_VEL
LIN {X 0,Y 148.01,Z 402.485,A -85,B 0,C 180,E1 -25436.702,E2 -25436.702} C_VEL
LIN {X 0,Y 145.224,Z 414.448,A -85,B 0,C 180,E1 -25438.654,E2 -25438.654} C_VEL
LIN {X 0,Y 141.971,Z 425.811,A -85,B 0,C 180,E1 -25441.143,E2 -25441.143} C_VEL
LIN {X 0,Y 138.571,Z 436.047,A -85,B 0,C 180,E1 -25444.061,E2 -25444.061} C_VEL
LIN {X 0,Y 135.339,Z 444.448,A -85,B 0,C 180,E1 -25447.081,E2 -25447.081} C_VEL
LIN {X 0,Y 132.143,Z 452.197,A -85,B 0,C 180,E1 -25450.587,E2 -25450.587} C_VEL
LIN {X 0,Y 128.816,Z 459.78,A -85,B 0,C 180,E1 -25454.982,E2 -25454.982} C_VEL
LIN {X 0,Y 126.549,Z 464.977,A -85,B 0,C 180,E1 -25458.793,E2 -25458.793} C_VEL
LIN {X 0,Y 124.456,Z 470.017,A -85,B 0,C 180,E1 -25463.517,E2 -25463.517} C_VEL
LIN {X 0,Y 122.852,Z 473.974,A -85,B 0,C 180,E1 -25468.362,E2 -25468.362} C_VEL
LIN {X 0,Y 122.06,Z 476.903,A -85,B 0,C 180,E1 -25473.302,E2 -25473.302} C_VEL
LIN {X 0,Y 122.03,Z 478.291,A -85,B 0,C 180,E1 -25476.615,E2 -25476.615} C_VEL
LIN {X 0,Y 122.674,Z 479.949,A -85,B 0,C 180,E1 -25483.249,E2 -25483.249} C_VEL
LIN {X 0,Y 123.439,Z 480.198,A -85,B 0,C 180,E1 -25486.54,E2 -25486.54} C_VEL
LIN {X 0,Y 125.946,Z 479.465,A -85,B 0,C 180,E1 -25492.993,E2 -25492.993} C_VEL
LIN {X 0,Y 127.698,Z 478.52,A -85,B 0,C 180,E1 -25496.123,E2 -25496.123} C_VEL
LIN {X 0,Y 131.312,Z 476.029,A -85,B 0,C 180,E1 -25501.089,E2 -25501.089} C_VEL
LIN {X 0,Y 136.277,Z 471.74,A -85,B 0,C 180,E1 -25506.376,E2 -25506.376} C_VEL
LIN {X 0,Y 140.974,Z 467.025,A -85,B 0,C 180,E1 -25510.398,E2 -25510.398} C_VEL
LIN {X 0,Y 146.263,Z 461.018,A -85,B 0,C 180,E1 -25514.164,E2 -25514.164} C_VEL
LIN {X 0,Y 152.068,Z 453.478,A -85,B 0,C 180,E1 -25517.685,E2 -25517.685} C_VEL
LIN {X 0,Y 157.197,Z 445.744,A -85,B 0,C 180,E1 -25520.433,E2 -25520.433} C_VEL
LIN {X 0,Y 162.59,Z 436.124,A -85,B 0,C 180,E1 -25523.096,E2 -25523.096} C_VEL
LIN {X 0,Y 167.653,Z 425.416,A -85,B 0,C 180,E1 -25525.354,E2 -25525.354} C_VEL
LIN {X 0,Y 171.677,Z 414.956,A -85,B 0,C 180,E1 -25527.057,E2 -25527.057} C_VEL
